Yaskawa INFORM job: DEMO_ROOF_UPPER_0625_3PAINT_68.JBI

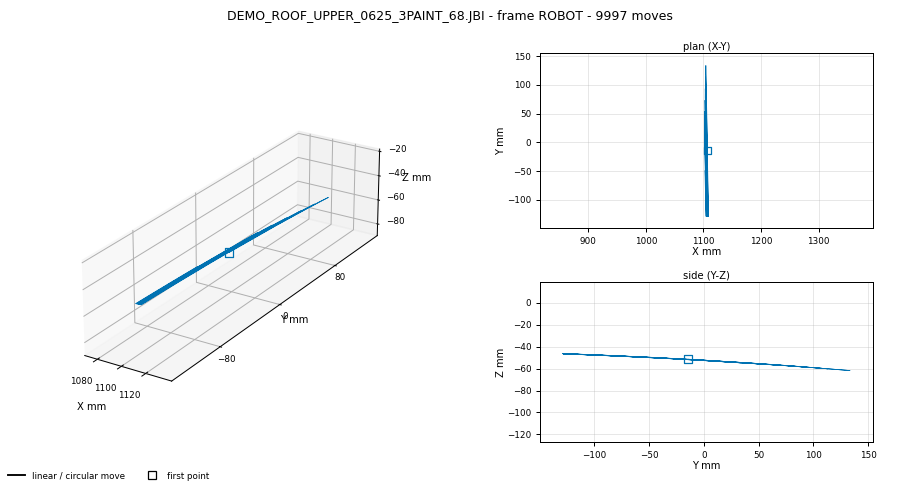
[picture p0: tool path of DEMO_ROOF_UPPER_0625_3PAINT_68.JBI in frame ROBOT, 9997 of 9997 moves have a stored position in this frame; points joined in program order, loops and branches not executed]
/JOB
//NAME DEMO_ROOF_UPPER_0625_3PAINT68
//POS
///NPOS 9997,0,0,0,0,0
///TOOL 0
///USER 0
///POSTYPE ROBOT
///RECTAN
///RCONF 1,0,0,0,0,0,0,0,0,0,0,0,0,0,0,0,0,0,0,0,0,0,0,0
C00000=1106.941,-14.112,-51.375,179.831,6.217,149.173
C00001=1106.936,-13.863,-51.390,179.832,6.222,149.174
C00002=1106.931,-13.614,-51.403,179.832,6.226,149.175
C00003=1106.926,-13.363,-51.417,179.833,6.230,149.176
C00004=1106.921,-13.114,-51.431,179.833,6.235,149.177
C00005=1106.916,-12.865,-51.445,179.834,6.239,149.177
C00006=1106.911,-12.615,-51.459,179.834,6.244,149.178
C00007=1106.906,-12.365,-51.472,179.835,6.249,149.179
C00008=1106.901,-12.115,-51.486,179.836,6.253,149.180
C00009=1106.896,-11.866,-51.500,179.836,6.258,149.181
C00010=1106.891,-11.617,-51.514,179.836,6.262,149.182
C00011=1106.886,-11.367,-51.529,179.837,6.266,149.183
C00012=1106.880,-11.117,-51.542,179.837,6.271,149.183
C00013=1106.876,-10.868,-51.555,179.838,6.276,149.184
C00014=1106.871,-10.618,-51.570,179.839,6.280,149.185
C00015=1106.865,-10.369,-51.584,179.839,6.285,149.186
C00016=1106.860,-10.120,-51.598,179.840,6.290,149.187
C00017=1106.855,-9.870,-51.612,179.840,6.294,149.188
C00018=1106.850,-9.619,-51.626,179.841,6.298,149.188
C00019=1106.845,-9.370,-51.640,179.841,6.303,149.189
C00020=1106.840,-9.121,-51.653,179.842,6.307,149.190
C00021=1106.835,-8.871,-51.668,179.842,6.312,149.191
C00022=1106.830,-8.622,-51.682,179.843,6.316,149.192
C00023=1106.825,-8.373,-51.696,179.844,6.321,149.193
C00024=1106.820,-8.123,-51.710,179.844,6.325,149.194
C00025=1106.815,-7.873,-51.724,179.844,6.330,149.194
C00026=1106.810,-7.623,-51.739,179.845,6.334,149.195
C00027=1106.804,-7.374,-51.753,179.846,6.339,149.196
C00028=1106.800,-7.125,-51.767,179.846,6.344,149.197
C00029=1106.795,-6.875,-51.781,179.847,6.348,149.198
C00030=1106.790,-6.625,-51.794,179.848,6.353,149.198
C00031=1106.785,-6.376,-51.808,179.848,6.357,149.199
C00032=1106.780,-6.126,-51.822,179.848,6.361,149.200
C00033=1106.775,-5.877,-51.837,179.849,6.366,149.201
C00034=1106.770,-5.627,-51.851,179.850,6.370,149.202
C00035=1106.764,-5.378,-51.865,179.850,6.375,149.203
C00036=1106.759,-5.128,-51.879,179.851,6.380,149.204
C00037=1106.756,-4.914,-51.892,179.851,6.383,149.204
C00038=1106.751,-4.700,-51.904,179.852,6.388,149.205
C00039=1106.747,-4.486,-51.916,179.852,6.391,149.206
C00040=1106.742,-4.271,-51.929,179.853,6.395,149.206
C00041=1106.738,-4.057,-51.941,179.853,6.399,149.207
C00042=1106.733,-3.844,-51.953,179.854,6.403,149.208
C00043=1106.729,-3.629,-51.966,179.854,6.406,149.209
C00044=1106.725,-3.415,-51.978,179.855,6.411,149.209
C00045=1106.720,-3.165,-51.992,179.856,6.415,149.210
C00046=1106.715,-2.916,-52.006,179.855,6.419,149.211
C00047=1106.709,-2.667,-52.020,179.856,6.424,149.212
C00048=1106.704,-2.417,-52.034,179.857,6.428,149.213
C00049=1106.699,-2.167,-52.049,179.857,6.433,149.213
C00050=1106.695,-1.918,-52.064,179.858,6.438,149.214
C00051=1106.690,-1.668,-52.078,179.859,6.442,149.215
C00052=1106.685,-1.419,-52.092,179.860,6.447,149.216
C00053=1106.679,-1.169,-52.107,179.860,6.452,149.217
C00054=1106.674,-0.920,-52.121,179.861,6.456,149.217
C00055=1106.669,-0.670,-52.135,179.862,6.461,149.218
C00056=1106.664,-0.421,-52.150,179.862,6.465,149.219
C00057=1106.659,-0.171,-52.165,179.862,6.469,149.220
C00058=1106.654,0.079,-52.179,179.863,6.474,149.221
C00059=1106.649,0.328,-52.193,179.864,6.478,149.222
C00060=1106.644,0.577,-52.208,179.865,6.483,149.222
C00061=1106.640,0.827,-52.222,179.865,6.487,149.223
C00062=1106.633,1.077,-52.237,179.866,6.492,149.224
C00063=1106.628,1.326,-52.251,179.866,6.497,149.225
C00064=1106.624,1.575,-52.266,179.867,6.501,149.226
C00065=1106.619,1.825,-52.280,179.868,6.506,149.227
C00066=1106.614,2.075,-52.295,179.868,6.511,149.227
C00067=1106.609,2.324,-52.310,179.869,6.515,149.228
C00068=1106.603,2.574,-52.325,179.870,6.520,149.229
C00069=1106.598,2.824,-52.339,179.870,6.524,149.230
C00070=1106.594,3.073,-52.354,179.871,6.529,149.231
C00071=1106.589,3.322,-52.368,179.872,6.533,149.231
C00072=1106.584,3.572,-52.382,179.872,6.538,149.232
C00073=1106.578,3.821,-52.398,179.873,6.543,149.233
C00074=1106.574,4.071,-52.412,179.873,6.547,149.234
C00075=1106.569,4.321,-52.427,179.874,6.551,149.235
C00076=1106.564,4.570,-52.442,179.874,6.556,149.236
C00077=1106.559,4.820,-52.456,179.875,6.560,149.237
C00078=1106.554,5.069,-52.471,179.875,6.565,149.237
C00079=1106.549,5.319,-52.486,179.876,6.569,149.238
C00080=1106.544,5.569,-52.500,179.877,6.574,149.239
C00081=1106.539,5.818,-52.515,179.878,6.579,149.240
C00082=1106.533,6.068,-52.530,179.878,6.584,149.241
C00083=1106.529,6.317,-52.545,179.879,6.588,149.241
C00084=1106.524,6.566,-52.559,179.880,6.593,149.242
C00085=1106.518,6.816,-52.575,179.880,6.597,149.243
C00086=1106.513,7.066,-52.589,179.881,6.602,149.244
C00087=1106.509,7.315,-52.604,179.882,6.606,149.245
C00088=1106.503,7.565,-52.619,179.882,6.611,149.246
C00089=1106.498,7.814,-52.634,179.883,6.616,149.247
C00090=1106.493,8.063,-52.648,179.883,6.620,149.247
C00091=1106.488,8.313,-52.664,179.884,6.625,149.248
C00092=1106.483,8.563,-52.678,179.885,6.630,149.249
C00093=1106.479,8.776,-52.691,179.885,6.634,149.250
C00094=1106.474,8.991,-52.704,179.886,6.638,149.251
C00095=1106.470,9.204,-52.716,179.886,6.642,149.251
C00096=1106.466,9.419,-52.729,179.886,6.645,149.252
C00097=1106.461,9.632,-52.742,179.887,6.649,149.253
C00098=1106.458,9.846,-52.755,179.887,6.653,149.254
C00099=1106.453,10.061,-52.768,179.888,6.657,149.254
C00100=1106.449,10.275,-52.781,179.888,6.661,149.255
C00101=1106.444,10.524,-52.795,179.888,6.666,149.256
C00102=1106.439,10.774,-52.811,179.889,6.670,149.257
C00103=1106.434,11.023,-52.826,179.889,6.674,149.258
C00104=1106.428,11.273,-52.841,179.890,6.679,149.259
C00105=1106.424,11.522,-52.856,179.890,6.683,149.259
C00106=1106.418,11.771,-52.871,179.891,6.688,149.260
C00107=1106.413,12.021,-52.886,179.891,6.692,149.261
C00108=1106.409,12.271,-52.901,179.891,6.697,149.262
C00109=1106.404,12.520,-52.917,179.892,6.701,149.263
C00110=1106.399,12.770,-52.931,179.892,6.705,149.264
C00111=1106.394,13.019,-52.946,179.893,6.709,149.265
C00112=1106.389,13.268,-52.961,179.893,6.714,149.265
C00113=1106.383,13.518,-52.976,179.894,6.719,149.266
C00114=1106.379,13.768,-52.991,179.894,6.723,149.267
C00115=1106.373,14.017,-53.007,179.895,6.727,149.268
C00116=1106.369,14.267,-53.022,179.895,6.732,149.269
C00117=1106.364,14.517,-53.037,179.895,6.736,149.270
C00118=1106.359,14.766,-53.052,179.896,6.740,149.270
C00119=1106.354,15.015,-53.068,179.897,6.745,149.271
C00120=1106.349,15.264,-53.083,179.897,6.749,149.272
C00121=1106.343,15.514,-53.098,179.897,6.753,149.273
C00122=1106.339,15.763,-53.113,179.898,6.758,149.274
C00123=1106.334,16.014,-53.129,179.899,6.762,149.274
C00124=1106.329,16.263,-53.143,179.900,6.767,149.275
C00125=1106.324,16.512,-53.159,179.900,6.771,149.276
C00126=1106.319,16.761,-53.174,179.901,6.775,149.277
C00127=1106.314,17.011,-53.190,179.901,6.780,149.278
C00128=1106.309,17.261,-53.204,179.901,6.784,149.279
C00129=1106.304,17.510,-53.220,179.902,6.788,149.279
C00130=1106.299,17.760,-53.235,179.903,6.793,149.280
C00131=1106.294,18.009,-53.250,179.903,6.798,149.281
C00132=1106.289,18.258,-53.266,179.904,6.801,149.282
C00133=1106.284,18.508,-53.281,179.904,6.806,149.283
C00134=1106.279,18.757,-53.297,179.905,6.811,149.284
C00135=1106.274,19.007,-53.313,179.905,6.814,149.284
C00136=1106.269,19.256,-53.328,179.906,6.819,149.285
C00137=1106.264,19.505,-53.343,179.907,6.823,149.286
C00138=1106.260,19.755,-53.359,179.907,6.828,149.287
C00139=1106.254,20.005,-53.374,179.908,6.831,149.287
C00140=1106.249,20.254,-53.390,179.908,6.836,149.288
C00141=1106.244,20.503,-53.405,179.909,6.841,149.289
C00142=1106.239,20.753,-53.421,179.909,6.844,149.290
C00143=1106.234,21.003,-53.436,179.910,6.849,149.291
C00144=1106.229,21.252,-53.451,179.911,6.853,149.291
C00145=1106.224,21.501,-53.467,179.912,6.858,149.292
C00146=1106.219,21.751,-53.483,179.912,6.862,149.293
C00147=1106.215,22.000,-53.498,179.913,6.866,149.294
C00148=1106.209,22.250,-53.513,179.914,6.871,149.294
C00149=1106.205,22.464,-53.527,179.914,6.874,149.295
C00150=1106.201,22.677,-53.540,179.915,6.878,149.296
C00151=1106.196,22.892,-53.554,179.915,6.881,149.296
C00152=1106.192,23.106,-53.567,179.915,6.885,149.297
C00153=1106.188,23.319,-53.580,179.916,6.889,149.298
C00154=1106.184,23.534,-53.594,179.917,6.892,149.298
C00155=1106.179,23.748,-53.607,179.917,6.896,149.299
C00156=1106.175,23.961,-53.620,179.918,6.899,149.300
C00157=1106.170,24.211,-53.636,179.919,6.904,149.300
C00158=1106.165,24.461,-53.652,179.919,6.908,149.301
C00159=1106.160,24.710,-53.667,179.920,6.912,149.302
C00160=1106.156,24.960,-53.683,179.921,6.916,149.302
C00161=1106.150,25.209,-53.698,179.921,6.921,149.303
C00162=1106.145,25.459,-53.714,179.922,6.925,149.304
C00163=1106.140,25.708,-53.730,179.922,6.929,149.305
C00164=1106.136,25.957,-53.745,179.923,6.934,149.306
C00165=1106.130,26.207,-53.761,179.924,6.937,149.306
C00166=1106.126,26.457,-53.777,179.924,6.942,149.307
C00167=1106.120,26.706,-53.793,179.926,6.946,149.308
C00168=1106.115,26.955,-53.809,179.927,6.950,149.308
C00169=1106.111,27.205,-53.824,179.927,6.954,149.309
C00170=1106.106,27.454,-53.840,179.928,6.959,149.310
C00171=1106.100,27.704,-53.855,179.929,6.963,149.311
C00172=1106.096,27.953,-53.872,179.929,6.967,149.311
C00173=1106.090,28.202,-53.888,179.930,6.971,149.312
C00174=1106.085,28.452,-53.903,179.931,6.975,149.313
C00175=1106.081,28.702,-53.919,179.931,6.979,149.313
C00176=1106.076,28.950,-53.935,179.932,6.984,149.314
C00177=1106.071,29.201,-53.951,179.933,6.988,149.315
C00178=1106.066,29.450,-53.966,179.934,6.992,149.316
C00179=1106.061,29.699,-53.983,179.934,6.996,149.316
C00180=1106.056,29.949,-53.999,179.935,7.000,149.317
C00181=1106.050,30.198,-54.014,179.936,7.005,149.318
C00182=1106.046,30.448,-54.031,179.936,7.008,149.318
C00183=1106.041,30.697,-54.046,179.937,7.013,149.319
C00184=1106.037,30.947,-54.062,179.938,7.017,149.320
C00185=1106.031,31.196,-54.078,179.939,7.022,149.321
C00186=1106.026,31.445,-54.094,179.940,7.025,149.321
C00187=1106.021,31.695,-54.110,179.941,7.029,149.322
C00188=1106.016,31.944,-54.126,179.942,7.034,149.323
C00189=1106.011,32.194,-54.142,179.942,7.037,149.323
C00190=1106.006,32.443,-54.158,179.943,7.042,149.324
C00191=1106.002,32.693,-54.174,179.944,7.046,149.325
C00192=1105.996,32.942,-54.191,179.944,7.050,149.326
C00193=1105.991,33.191,-54.206,179.945,7.054,149.326
C00194=1105.987,33.441,-54.223,179.946,7.058,149.327
C00195=1105.981,33.690,-54.238,179.947,7.063,149.327
C00196=1105.976,33.940,-54.254,179.948,7.066,149.328
C00197=1105.971,34.189,-54.271,179.948,7.071,149.329
C00198=1105.967,34.439,-54.287,179.950,7.075,149.330
C00199=1105.961,34.688,-54.303,179.950,7.079,149.330
C00200=1105.957,34.937,-54.320,179.951,7.083,149.331
C00201=1105.952,35.187,-54.335,179.952,7.087,149.332
C00202=1105.947,35.436,-54.352,179.953,7.092,149.332
C00203=1105.942,35.686,-54.367,179.954,7.095,149.333
C00204=1105.937,35.935,-54.384,179.955,7.099,149.334
C00205=1105.933,36.149,-54.398,179.955,7.103,149.334
C00206=1105.928,36.362,-54.412,179.956,7.106,149.335
C00207=1105.924,36.577,-54.426,179.957,7.110,149.335
C00208=1105.920,36.791,-54.439,179.958,7.114,149.336
C00209=1105.916,37.005,-54.454,179.958,7.117,149.336
C00210=1105.911,37.219,-54.467,179.959,7.121,149.337
C00211=1105.907,37.432,-54.482,179.960,7.124,149.338
C00212=1105.903,37.646,-54.495,179.960,7.127,149.338
C00213=1105.898,37.896,-54.512,179.961,7.132,149.339
C00214=1105.893,38.145,-54.528,179.962,7.136,149.340
C00215=1105.888,38.395,-54.544,179.963,7.140,149.340
C00216=1105.883,38.644,-54.560,179.964,7.144,149.341
C00217=1105.879,38.893,-54.577,179.965,7.148,149.341
C00218=1105.873,39.143,-54.594,179.966,7.152,149.342
C00219=1105.868,39.392,-54.610,179.967,7.156,149.343
C00220=1105.864,39.642,-54.627,179.968,7.160,149.343
C00221=1105.858,39.891,-54.642,179.969,7.164,149.344
C00222=1105.854,40.141,-54.659,179.970,7.169,149.345
C00223=1105.849,40.389,-54.675,179.971,7.172,149.345
C00224=1105.844,40.639,-54.691,179.972,7.176,149.346
C00225=1105.839,40.889,-54.708,179.973,7.180,149.347
C00226=1105.834,41.138,-54.725,179.974,7.185,149.347
C00227=1105.829,41.388,-54.741,179.974,7.188,149.348
C00228=1105.824,41.636,-54.758,179.975,7.193,149.348
C00229=1105.819,41.886,-54.774,179.977,7.197,149.349
C00230=1105.814,42.136,-54.791,179.977,7.200,149.350
C00231=1105.809,42.385,-54.807,179.978,7.205,149.350
C00232=1105.804,42.634,-54.824,179.979,7.209,149.351
C00233=1105.799,42.883,-54.840,179.981,7.213,149.352
C00234=1105.794,43.134,-54.857,179.981,7.216,149.352
C00235=1105.789,43.383,-54.873,179.982,7.221,149.353
C00236=1105.784,43.632,-54.890,179.983,7.225,149.353
C00237=1105.780,43.881,-54.906,179.984,7.229,149.354
C00238=1105.775,44.131,-54.924,179.985,7.233,149.355
C00239=1105.770,44.380,-54.940,179.986,7.237,149.355
C00240=1105.765,44.629,-54.957,179.987,7.241,149.356
C00241=1105.761,44.879,-54.973,179.988,7.245,149.357
C00242=1105.754,45.129,-54.989,179.989,7.249,149.357
C00243=1105.750,45.378,-55.006,179.990,7.253,149.358
C00244=1105.745,45.628,-55.023,179.991,7.257,149.359
C00245=1105.740,45.877,-55.040,179.992,7.261,149.359
C00246=1105.735,46.126,-55.056,179.993,7.265,149.360
C00247=1105.731,46.376,-55.073,179.994,7.269,149.360
C00248=1105.726,46.624,-55.089,179.995,7.273,149.361
C00249=1105.720,46.874,-55.107,179.996,7.277,149.362
C00250=1105.716,47.124,-55.123,179.997,7.281,149.362
C00251=1105.711,47.373,-55.140,179.998,7.285,149.363
C00252=1105.706,47.622,-55.157,179.999,7.289,149.363
C00253=1105.701,47.872,-55.174,180.000,7.293,149.364
C00254=1105.696,48.122,-55.191,-179.999,7.297,149.364
C00255=1105.691,48.371,-55.207,-179.997,7.301,149.365
C00256=1105.686,48.620,-55.224,-179.997,7.305,149.366
C00257=1105.681,48.870,-55.241,-179.996,7.309,149.366
C00258=1105.677,49.119,-55.258,-179.994,7.313,149.367
C00259=1105.672,49.367,-55.275,-179.993,7.317,149.367
C00260=1105.667,49.617,-55.292,-179.993,7.321,149.368
C00261=1105.663,49.831,-55.306,-179.991,7.325,149.369
C00262=1105.658,50.045,-55.320,-179.990,7.328,149.369
C00263=1105.654,50.259,-55.335,-179.990,7.331,149.370
C00264=1105.650,50.473,-55.350,-179.989,7.334,149.370
C00265=1105.646,50.687,-55.364,-179.987,7.338,149.371
C00266=1105.642,50.900,-55.378,-179.987,7.342,149.371
C00267=1105.637,51.114,-55.393,-179.986,7.345,149.372
C00268=1105.633,51.328,-55.408,-179.985,7.348,149.372
C00269=1105.628,51.577,-55.424,-179.984,7.352,149.373
C00270=1105.623,51.827,-55.442,-179.982,7.356,149.373
C00271=1105.619,52.075,-55.459,-179.982,7.360,149.374
C00272=1105.613,52.325,-55.476,-179.981,7.364,149.374
C00273=1105.609,52.575,-55.493,-179.979,7.368,149.375
C00274=1105.604,52.825,-55.510,-179.978,7.372,149.376
C00275=1105.599,53.073,-55.527,-179.978,7.376,149.376
C00276=1105.594,53.322,-55.544,-179.976,7.380,149.377
C00277=1105.589,53.572,-55.561,-179.975,7.384,149.377
C00278=1105.584,53.822,-55.578,-179.974,7.388,149.378
C00279=1105.579,54.071,-55.596,-179.972,7.392,149.378
C00280=1105.575,54.320,-55.613,-179.972,7.396,149.379
C00281=1105.569,54.570,-55.630,-179.970,7.400,149.379
C00282=1105.564,54.819,-55.646,-179.969,7.404,149.380
C00283=1105.559,55.068,-55.664,-179.968,7.408,149.381
C00284=1105.555,55.318,-55.681,-179.967,7.411,149.381
C00285=1105.550,55.567,-55.698,-179.966,7.416,149.382
C00286=1105.545,55.816,-55.716,-179.965,7.420,149.382
C00287=1105.540,56.066,-55.733,-179.964,7.424,149.383
C00288=1105.535,56.316,-55.750,-179.963,7.427,149.383
C00289=1105.530,56.564,-55.767,-179.962,7.431,149.384
C00290=1105.525,56.814,-55.785,-179.960,7.436,149.385
C00291=1105.520,57.063,-55.803,-179.959,7.439,149.385
C00292=1105.516,57.313,-55.819,-179.958,7.444,149.386
C00293=1105.510,57.562,-55.836,-179.957,7.447,149.386
C00294=1105.506,57.811,-55.854,-179.956,7.451,149.387
C00295=1105.501,58.061,-55.871,-179.954,7.455,149.387
C00296=1105.496,58.310,-55.889,-179.953,7.459,149.388
C00297=1105.492,58.560,-55.906,-179.952,7.463,149.388
C00298=1105.487,58.809,-55.924,-179.951,7.467,149.389
C00299=1105.481,59.059,-55.941,-179.949,7.471,149.389
C00300=1105.477,59.307,-55.958,-179.948,7.475,149.390
C00301=1105.471,59.557,-55.975,-179.947,7.479,149.391
C00302=1105.467,59.806,-55.993,-179.946,7.482,149.391
C00303=1105.461,60.056,-56.011,-179.945,7.486,149.392
C00304=1105.457,60.304,-56.028,-179.944,7.491,149.392
C00305=1105.452,60.554,-56.045,-179.942,7.495,149.393
C00306=1105.447,60.803,-56.063,-179.941,7.499,149.393
C00307=1105.443,61.053,-56.080,-179.940,7.502,149.394
C00308=1105.438,61.302,-56.098,-179.939,7.506,149.394
C00309=1105.432,61.552,-56.115,-179.937,7.510,149.395
C00310=1105.428,61.801,-56.133,-179.936,7.514,149.396
C00311=1105.423,62.050,-56.150,-179.935,7.518,149.396
C00312=1105.418,62.300,-56.168,-179.934,7.522,149.397
C00313=1105.413,62.549,-56.186,-179.933,7.526,149.397
C00314=1105.408,62.799,-56.203,-179.932,7.530,149.398
C00315=1105.404,63.047,-56.220,-179.930,7.534,149.398
C00316=1105.399,63.297,-56.238,-179.929,7.538,149.399
C00317=1105.394,63.511,-56.253,-179.928,7.541,149.399
C00318=1105.391,63.724,-56.268,-179.927,7.544,149.400
C00319=1105.386,63.938,-56.283,-179.925,7.548,149.400
C00320=1105.382,64.152,-56.298,-179.925,7.551,149.401
C00321=1105.378,64.366,-56.314,-179.924,7.555,149.401
C00322=1105.373,64.580,-56.329,-179.923,7.558,149.401
C00323=1105.370,64.793,-56.344,-179.921,7.562,149.402
C00324=1105.365,65.007,-56.359,-179.920,7.565,149.402
C00325=1105.360,65.256,-56.377,-179.919,7.569,149.403
C00326=1105.356,65.505,-56.395,-179.917,7.573,149.403
C00327=1105.351,65.754,-56.412,-179.917,7.576,149.404
C00328=1105.346,66.004,-56.430,-179.915,7.580,149.404
C00329=1105.341,66.254,-56.448,-179.914,7.584,149.405
C00330=1105.336,66.503,-56.466,-179.913,7.589,149.406
C00331=1105.331,66.752,-56.484,-179.911,7.592,149.406
C00332=1105.326,67.002,-56.501,-179.910,7.597,149.407
C00333=1105.321,67.251,-56.519,-179.909,7.600,149.407
C00334=1105.316,67.500,-56.537,-179.908,7.604,149.408
C00335=1105.312,67.749,-56.555,-179.906,7.608,149.408
C00336=1105.307,67.998,-56.573,-179.905,7.612,149.409
C00337=1105.302,68.247,-56.591,-179.903,7.616,149.409
C00338=1105.297,68.497,-56.608,-179.902,7.620,149.410
C00339=1105.292,68.746,-56.626,-179.901,7.624,149.410
C00340=1105.288,68.996,-56.644,-179.900,7.628,149.411
C00341=1105.283,69.245,-56.662,-179.899,7.631,149.411
C00342=1105.278,69.494,-56.680,-179.897,7.635,149.412
C00343=1105.273,69.744,-56.698,-179.896,7.640,149.412
C00344=1105.268,69.993,-56.716,-179.894,7.644,149.413
C00345=1105.263,70.242,-56.734,-179.893,7.647,149.413
C00346=1105.259,70.491,-56.752,-179.892,7.652,149.414
C00347=1105.254,70.740,-56.770,-179.891,7.655,149.414
C00348=1105.249,70.990,-56.788,-179.889,7.659,149.415
C00349=1105.244,71.239,-56.806,-179.888,7.663,149.415
C00350=1105.239,71.489,-56.824,-179.886,7.667,149.416
C00351=1105.235,71.738,-56.842,-179.885,7.671,149.416
C00352=1105.230,71.987,-56.860,-179.884,7.675,149.417
C00353=1105.225,72.236,-56.878,-179.882,7.679,149.417
C00354=1105.220,72.486,-56.897,-179.881,7.683,149.418
C00355=1105.216,72.735,-56.915,-179.880,7.686,149.418
C00356=1105.210,72.985,-56.933,-179.878,7.690,149.419
C00357=1105.205,73.234,-56.951,-179.877,7.694,149.419
C00358=1105.200,73.483,-56.969,-179.876,7.698,149.420
C00359=1105.196,73.733,-56.988,-179.874,7.702,149.420
C00360=1105.191,73.982,-57.006,-179.873,7.706,149.421
C00361=1105.186,74.231,-57.023,-179.872,7.711,149.421
C00362=1105.181,74.480,-57.041,-179.870,7.714,149.422
C00363=1105.176,74.729,-57.060,-179.868,7.718,149.422
C00364=1105.172,74.979,-57.079,-179.867,7.721,149.423
C00365=1105.166,75.228,-57.097,-179.866,7.726,149.423
C00366=1105.162,75.477,-57.115,-179.865,7.730,149.424
C00367=1105.157,75.727,-57.133,-179.863,7.734,149.424
C00368=1105.152,75.977,-57.151,-179.862,7.738,149.425
C00369=1105.148,76.225,-57.170,-179.860,7.742,149.425
C00370=1105.143,76.474,-57.188,-179.859,7.746,149.426
C00371=1105.137,76.724,-57.207,-179.857,7.750,149.426
C00372=1105.133,76.974,-57.225,-179.856,7.754,149.427
C00373=1105.128,77.187,-57.241,-179.855,7.757,149.427
C00374=1105.124,77.400,-57.256,-179.854,7.760,149.428
C00375=1105.121,77.614,-57.272,-179.853,7.763,149.428
C00376=1105.116,77.828,-57.288,-179.853,7.767,149.429
C00377=1105.112,78.041,-57.303,-179.852,7.770,149.429
C00378=1105.108,78.255,-57.320,-179.851,7.773,149.430
C00379=1105.104,78.468,-57.335,-179.851,7.775,149.430
C00380=1105.100,78.683,-57.351,-179.850,7.778,149.431
C00381=1105.095,78.932,-57.369,-179.848,7.783,149.431
C00382=1105.091,79.180,-57.388,-179.848,7.786,149.432
C00383=1105.085,79.430,-57.407,-179.846,7.790,149.432
C00384=1105.081,79.680,-57.425,-179.846,7.794,149.433
C00385=1105.076,79.928,-57.444,-179.844,7.797,149.433
C00386=1105.071,80.177,-57.462,-179.844,7.801,149.434
C00387=1105.066,80.428,-57.481,-179.842,7.805,149.434
C00388=1105.061,80.676,-57.499,-179.842,7.808,149.435
C00389=1105.056,80.925,-57.517,-179.840,7.812,149.436
C00390=1105.052,81.175,-57.537,-179.839,7.816,149.436
C00391=1105.047,81.424,-57.555,-179.838,7.820,149.437
C00392=1105.042,81.673,-57.573,-179.837,7.824,149.437
C00393=1105.037,81.923,-57.593,-179.836,7.827,149.438
C00394=1105.032,82.172,-57.611,-179.835,7.831,149.438
C00395=1105.028,82.421,-57.629,-179.834,7.834,149.439
C00396=1105.023,82.671,-57.648,-179.833,7.839,149.439
C00397=1105.018,82.919,-57.667,-179.832,7.842,149.440
C00398=1105.014,83.169,-57.685,-179.831,7.846,149.441
C00399=1105.008,83.419,-57.704,-179.830,7.849,149.441
C00400=1105.003,83.667,-57.722,-179.829,7.853,149.442
C00401=1104.999,83.917,-57.741,-179.827,7.857,149.442
C00402=1104.994,84.166,-57.760,-179.826,7.861,149.443
C00403=1104.989,84.415,-57.778,-179.825,7.865,149.443
C00404=1104.984,84.665,-57.798,-179.824,7.868,149.444
C00405=1104.979,84.913,-57.816,-179.823,7.872,149.444
C00406=1104.975,85.163,-57.835,-179.822,7.876,149.445
C00407=1104.970,85.412,-57.854,-179.821,7.879,149.445
C00408=1104.965,85.661,-57.872,-179.819,7.884,149.446
C00409=1104.960,85.911,-57.892,-179.819,7.887,149.446
C00410=1104.955,86.160,-57.910,-179.817,7.891,149.447
C00411=1104.951,86.409,-57.929,-179.816,7.895,149.448
C00412=1104.946,86.658,-57.948,-179.815,7.898,149.448
C00413=1104.942,86.908,-57.966,-179.814,7.902,149.449
C00414=1104.936,87.157,-57.986,-179.813,7.906,149.449
C00415=1104.931,87.406,-58.004,-179.812,7.910,149.450
C00416=1104.927,87.656,-58.023,-179.810,7.914,149.450
C00417=1104.922,87.904,-58.042,-179.809,7.917,149.451
C00418=1104.917,88.154,-58.061,-179.808,7.921,149.451
C00419=1104.912,88.403,-58.080,-179.806,7.925,149.452
C00420=1104.908,88.652,-58.099,-179.805,7.928,149.452
C00421=1104.903,88.902,-58.117,-179.804,7.932,149.453
C00422=1104.898,89.151,-58.137,-179.803,7.936,149.453
C00423=1104.893,89.400,-58.156,-179.802,7.940,149.454
C00424=1104.889,89.649,-58.175,-179.801,7.944,149.454
C00425=1104.884,89.898,-58.193,-179.799,7.947,149.455
C00426=1104.879,90.148,-58.213,-179.798,7.951,149.455
C00427=1104.874,90.397,-58.232,-179.797,7.955,149.456
C00428=1104.870,90.646,-58.251,-179.795,7.959,149.456
C00429=1104.865,90.859,-58.267,-179.794,7.962,149.457
C00430=1104.861,91.074,-58.283,-179.793,7.965,149.457
C00431=1104.857,91.287,-58.300,-179.792,7.968,149.458
C00432=1104.853,91.501,-58.316,-179.791,7.971,149.458
C00433=1104.849,91.714,-58.333,-179.790,7.975,149.458
C00434=1104.845,91.928,-58.349,-179.789,7.978,149.459
C00435=1104.841,92.140,-58.365,-179.788,7.981,149.459
C00436=1104.836,92.355,-58.382,-179.787,7.984,149.460
C00437=1104.831,92.603,-58.401,-179.785,7.988,149.460
C00438=1104.827,92.853,-58.420,-179.784,7.991,149.461
C00439=1104.823,93.102,-58.439,-179.783,7.995,149.461
C00440=1104.817,93.351,-58.459,-179.782,8.000,149.462
C00441=1104.812,93.601,-58.478,-179.780,8.003,149.462
C00442=1104.808,93.850,-58.496,-179.779,8.007,149.463
C00443=1104.803,94.099,-58.516,-179.777,8.010,149.463
C00444=1104.798,94.348,-58.535,-179.776,8.014,149.463
C00445=1104.794,94.597,-58.554,-179.775,8.019,149.464
C00446=1104.788,94.846,-58.574,-179.774,8.022,149.464
C00447=1104.784,95.096,-58.593,-179.772,8.026,149.465
C00448=1104.780,95.345,-58.612,-179.770,8.030,149.465
C00449=1104.774,95.594,-58.632,-179.769,8.033,149.466
C00450=1104.769,95.844,-58.651,-179.768,8.036,149.466
C00451=1104.764,96.092,-58.671,-179.766,8.040,149.467
C00452=1104.760,96.342,-58.690,-179.765,8.045,149.467
C00453=1104.755,96.591,-58.709,-179.764,8.048,149.468
C00454=1104.750,96.840,-58.729,-179.763,8.052,149.468
C00455=1104.746,97.089,-58.748,-179.761,8.056,149.469
C00456=1104.741,97.338,-58.767,-179.759,8.059,149.469
C00457=1104.736,97.588,-58.787,-179.758,8.063,149.469
C00458=1104.731,97.837,-58.806,-179.757,8.066,149.470
C00459=1104.726,98.086,-58.825,-179.755,8.070,149.470
C00460=1104.722,98.336,-58.845,-179.754,8.074,149.471
C00461=1104.717,98.585,-58.864,-179.752,8.078,149.471
C00462=1104.712,98.834,-58.883,-179.751,8.081,149.472
C00463=1104.707,99.083,-58.904,-179.749,8.085,149.472
C00464=1104.703,99.332,-58.923,-179.748,8.089,149.473
C00465=1104.698,99.581,-58.942,-179.746,8.093,149.473
C00466=1104.693,99.831,-58.962,-179.745,8.097,149.473
C00467=1104.688,100.080,-58.982,-179.744,8.100,149.474
C00468=1104.683,100.329,-59.001,-179.742,8.104,149.474
C00469=1104.679,100.578,-59.021,-179.740,8.108,149.475
C00470=1104.675,100.827,-59.040,-179.739,8.111,149.475
C00471=1104.669,101.076,-59.060,-179.737,8.114,149.475
C00472=1104.665,101.326,-59.079,-179.736,8.118,149.476
C00473=1104.660,101.575,-59.099,-179.734,8.122,149.476
C00474=1104.655,101.824,-59.119,-179.733,8.126,149.477
C00475=1104.650,102.073,-59.139,-179.731,8.130,149.477
C00476=1104.645,102.323,-59.158,-179.729,8.134,149.478
C00477=1104.641,102.572,-59.178,-179.728,8.137,149.478
C00478=1104.636,102.820,-59.198,-179.726,8.140,149.478
C00479=1104.632,103.070,-59.217,-179.725,8.144,149.479
C00480=1104.627,103.319,-59.237,-179.723,8.148,149.479
C00481=1104.622,103.568,-59.257,-179.722,8.152,149.480
C00482=1104.617,103.817,-59.276,-179.721,8.155,149.480
C00483=1104.612,104.067,-59.296,-179.718,8.159,149.480
C00484=1104.608,104.316,-59.316,-179.717,8.162,149.481
C00485=1104.604,104.529,-59.334,-179.715,8.165,149.481
C00486=1104.599,104.743,-59.349,-179.714,8.169,149.481
C00487=1104.595,104.957,-59.367,-179.712,8.172,149.482
C00488=1104.591,105.170,-59.384,-179.711,8.175,149.482
C00489=1104.587,105.383,-59.401,-179.710,8.178,149.482
C00490=1104.583,105.597,-59.417,-179.708,8.181,149.483
C00491=1104.579,105.810,-59.435,-179.707,8.184,149.483
C00492=1104.575,106.024,-59.452,-179.706,8.187,149.483
C00493=1104.570,106.272,-59.472,-179.704,8.191,149.484
C00494=1104.566,106.522,-59.491,-179.702,8.195,149.484
C00495=1104.561,106.771,-59.512,-179.700,8.198,149.484
C00496=1104.556,107.020,-59.531,-179.699,8.202,149.485
C00497=1104.552,107.269,-59.552,-179.697,8.205,149.485
C00498=1104.547,107.518,-59.571,-179.696,8.209,149.485
C00499=1104.542,107.767,-59.591,-179.694,8.213,149.486
C00500=1104.537,108.017,-59.612,-179.692,8.216,149.486
C00501=1104.532,108.266,-59.632,-179.690,8.220,149.486
C00502=1104.527,108.515,-59.652,-179.688,8.223,149.487
C00503=1104.523,108.764,-59.672,-179.687,8.227,149.487
C00504=1104.518,109.014,-59.692,-179.685,8.230,149.487
C00505=1104.513,109.262,-59.712,-179.683,8.234,149.487
C00506=1104.508,109.512,-59.731,-179.682,8.237,149.488
C00507=1104.504,109.761,-59.752,-179.680,8.241,149.488
C00508=1104.500,110.010,-59.772,-179.678,8.245,149.489
C00509=1104.494,110.259,-59.792,-179.676,8.248,149.489
C00510=1104.490,110.508,-59.813,-179.674,8.251,149.489
C00511=1104.485,110.757,-59.833,-179.673,8.255,149.489
C00512=1104.480,111.006,-59.852,-179.671,8.258,149.490
C00513=1104.475,111.255,-59.873,-179.669,8.262,149.490
C00514=1104.471,111.504,-59.893,-179.667,8.266,149.490
C00515=1104.466,111.754,-59.913,-179.666,8.268,149.491
C00516=1104.461,112.003,-59.934,-179.664,8.272,149.491
C00517=1104.457,112.252,-59.954,-179.662,8.276,149.491
C00518=1104.452,112.501,-59.974,-179.661,8.279,149.492
C00519=1104.448,112.750,-59.994,-179.659,8.282,149.492
C00520=1104.442,113.000,-60.015,-179.657,8.286,149.492
C00521=1104.438,113.249,-60.036,-179.656,8.289,149.493
C00522=1104.433,113.498,-60.055,-179.654,8.293,149.493
C00523=1104.429,113.747,-60.076,-179.652,8.296,149.493
C00524=1104.423,113.996,-60.096,-179.651,8.299,149.494
C00525=1104.419,114.245,-60.117,-179.649,8.303,149.494
C00526=1104.414,114.494,-60.136,-179.647,8.307,149.494
C00527=1104.409,114.743,-60.157,-179.646,8.309,149.494
C00528=1104.404,114.992,-60.178,-179.644,8.313,149.495
C00529=1104.400,115.241,-60.198,-179.642,8.317,149.495
C00530=1104.395,115.490,-60.218,-179.641,8.319,149.495
C00531=1104.390,115.740,-60.239,-179.639,8.323,149.496
C00532=1104.385,115.989,-60.259,-179.637,8.327,149.496
C00533=1104.381,116.238,-60.279,-179.635,8.329,149.496
C00534=1104.376,116.487,-60.300,-179.633,8.333,149.496
C00535=1104.371,116.736,-60.321,-179.632,8.337,149.497
C00536=1104.367,116.985,-60.341,-179.630,8.340,149.497
C00537=1104.362,117.235,-60.362,-179.628,8.343,149.497
C00538=1104.357,117.483,-60.382,-179.627,8.347,149.498
C00539=1104.353,117.732,-60.403,-179.625,8.350,149.498
C00540=1104.348,117.982,-60.424,-179.623,8.353,149.498
C00541=1104.344,118.195,-60.440,-179.622,8.356,149.498
C00542=1104.340,118.408,-60.459,-179.621,8.359,149.499
C00543=1104.336,118.622,-60.476,-179.619,8.362,149.499
C00544=1104.332,118.835,-60.494,-179.617,8.365,149.499
C00545=1104.328,119.049,-60.512,-179.616,8.368,149.500
C00546=1104.324,119.262,-60.530,-179.614,8.371,149.500
C00547=1104.320,119.476,-60.546,-179.613,8.373,149.500
C00548=1104.316,119.688,-60.564,-179.612,8.376,149.500
C00549=1104.311,119.938,-60.586,-179.609,8.380,149.500
C00550=1104.307,120.187,-60.606,-179.608,8.383,149.501
C00551=1104.302,120.436,-60.627,-179.606,8.386,149.501
C00552=1104.297,120.685,-60.647,-179.604,8.390,149.501
C00553=1104.292,120.935,-60.668,-179.603,8.393,149.502
C00554=1104.288,121.183,-60.689,-179.601,8.396,149.502
C00555=1104.283,121.432,-60.709,-179.599,8.400,149.502
C00556=1104.278,121.681,-60.731,-179.598,8.402,149.502
C00557=1104.274,121.930,-60.751,-179.596,8.406,149.503
C00558=1104.269,122.179,-60.772,-179.594,8.410,149.503
C00559=1104.264,122.428,-60.792,-179.593,8.413,149.503
C00560=1104.260,122.678,-60.814,-179.591,8.416,149.504
C00561=1104.255,122.927,-60.834,-179.589,8.420,149.504
C00562=1104.250,123.176,-60.856,-179.588,8.423,149.504
C00563=1104.246,123.425,-60.876,-179.585,8.426,149.505
C00564=1104.241,123.674,-60.897,-179.583,8.430,149.505
C00565=1104.236,123.923,-60.917,-179.582,8.434,149.505
C00566=1104.231,124.172,-60.938,-179.580,8.436,149.505
C00567=1104.227,124.422,-60.960,-179.578,8.440,149.506
C00568=1104.222,124.670,-60.981,-179.577,8.444,149.506
C00569=1104.217,124.920,-61.002,-179.575,8.446,149.506
C00570=1104.213,125.169,-61.022,-179.573,8.450,149.507
C00571=1104.208,125.417,-61.044,-179.571,8.453,149.507
C00572=1104.203,125.666,-61.064,-179.570,8.456,149.507
C00573=1104.199,125.916,-61.086,-179.568,8.460,149.507
C00574=1104.194,126.165,-61.107,-179.566,8.463,149.508
C00575=1104.190,126.414,-61.128,-179.565,8.466,149.508
C00576=1104.184,126.663,-61.149,-179.562,8.470,149.508
C00577=1104.180,126.911,-61.170,-179.561,8.474,149.509
C00578=1104.176,127.161,-61.191,-179.559,8.476,149.509
C00579=1104.170,127.411,-61.212,-179.557,8.480,149.509
C00580=1104.166,127.659,-61.233,-179.555,8.483,149.509
C00581=1104.161,127.908,-61.254,-179.554,8.486,149.510
C00582=1104.156,128.157,-61.275,-179.552,8.490,149.510
C00583=1104.152,128.406,-61.296,-179.550,8.493,149.510
C00584=1104.147,128.656,-61.317,-179.549,8.496,149.510
C00585=1104.142,128.904,-61.339,-179.547,8.500,149.511
C00586=1104.137,129.154,-61.360,-179.545,8.503,149.511
C00587=1104.133,129.402,-61.381,-179.544,8.506,149.511
C00588=1104.129,129.652,-61.403,-179.541,8.510,149.512
C00589=1104.124,129.901,-61.424,-179.540,8.513,149.512
C00590=1104.119,130.150,-61.445,-179.538,8.517,149.512
C00591=1104.114,130.398,-61.466,-179.536,8.520,149.512
C00592=1104.110,130.648,-61.488,-179.534,8.523,149.513
C00593=1104.105,130.897,-61.509,-179.533,8.527,149.513
C00594=1104.101,131.146,-61.530,-179.531,8.530,149.513
C00595=1104.096,131.395,-61.552,-179.529,8.533,149.514
C00596=1104.091,131.644,-61.573,-179.527,8.537,149.514
C00597=1104.087,131.878,-61.592,-179.526,8.539,149.514
C00598=1104.083,132.113,-61.613,-179.524,8.543,149.514
C00599=1104.078,132.348,-61.633,-179.523,8.546,149.515
C00600=1104.073,132.582,-61.653,-179.520,8.550,149.515
C00601=1104.069,132.816,-61.673,-179.519,8.552,149.515
C00602=1104.065,133.051,-61.694,-179.517,8.556,149.515
C00603=1104.060,133.285,-61.714,-179.516,8.559,149.516
C00604=1104.056,133.520,-61.734,-179.514,8.562,149.516
C00605=1103.825,123.405,-60.927,-179.583,8.428,149.504
C00606=1103.830,123.156,-60.906,-179.585,8.424,149.504
C00607=1103.835,122.908,-60.885,-179.586,8.421,149.503
C00608=1103.839,122.658,-60.864,-179.588,8.418,149.503
C00609=1103.844,122.409,-60.843,-179.590,8.414,149.503
C00610=1103.849,122.160,-60.822,-179.591,8.411,149.503
C00611=1103.853,121.911,-60.802,-179.593,8.408,149.502
C00612=1103.858,121.662,-60.781,-179.595,8.404,149.502
C00613=1103.863,121.413,-60.760,-179.596,8.401,149.502
C00614=1103.868,121.164,-60.739,-179.599,8.398,149.502
C00615=1103.872,120.915,-60.718,-179.600,8.394,149.501
C00616=1103.877,120.666,-60.697,-179.602,8.391,149.501
C00617=1103.881,120.416,-60.677,-179.604,8.388,149.501
C00618=1103.886,120.167,-60.656,-179.605,8.384,149.500
C00619=1103.891,119.918,-60.635,-179.607,8.381,149.500
C00620=1103.895,119.669,-60.615,-179.609,8.378,149.500
C00621=1103.900,119.420,-60.594,-179.611,8.374,149.500
C00622=1103.907,119.061,-60.564,-179.613,8.370,149.499
C00623=1103.914,118.704,-60.535,-179.615,8.365,149.499
C00624=1103.921,118.345,-60.505,-179.618,8.360,149.498
C00625=1103.928,117.987,-60.476,-179.620,8.355,149.498
C00626=1103.932,117.738,-60.455,-179.622,8.352,149.498
C00627=1103.937,117.488,-60.434,-179.624,8.349,149.497
C00628=1103.942,117.239,-60.414,-179.626,8.345,149.497
C00629=1103.946,116.990,-60.394,-179.627,8.342,149.497
C00630=1103.951,116.741,-60.373,-179.629,8.338,149.496
C00631=1103.956,116.492,-60.352,-179.631,8.335,149.496
C00632=1103.960,116.243,-60.332,-179.632,8.332,149.496
C00633=1103.965,115.994,-60.311,-179.634,8.328,149.496
C00634=1103.970,115.745,-60.291,-179.636,8.324,149.495
C00635=1103.974,115.496,-60.270,-179.637,8.322,149.495
C00636=1103.980,115.246,-60.250,-179.639,8.318,149.494
C00637=1103.984,114.997,-60.230,-179.641,8.314,149.494
C00638=1103.989,114.748,-60.209,-179.642,8.312,149.494
C00639=1103.993,114.499,-60.189,-179.644,8.308,149.494
C00640=1103.998,114.250,-60.168,-179.646,8.304,149.493
C00641=1104.003,114.001,-60.148,-179.647,8.302,149.493
C00642=1104.007,113.752,-60.128,-179.649,8.298,149.493
C00643=1104.013,113.502,-60.107,-179.651,8.294,149.492
C00644=1104.017,113.253,-60.087,-179.652,8.291,149.492
C00645=1104.021,113.005,-60.066,-179.654,8.288,149.492
C00646=1104.026,112.755,-60.047,-179.656,8.284,149.492
C00647=1104.031,112.506,-60.026,-179.657,8.281,149.491
C00648=1104.036,112.257,-60.005,-179.659,8.277,149.491
C00649=1104.041,112.008,-59.985,-179.661,8.274,149.490
C00650=1104.046,111.759,-59.966,-179.662,8.271,149.490
C00651=1104.050,111.510,-59.945,-179.664,8.267,149.490
C00652=1104.055,111.261,-59.924,-179.666,8.263,149.490
C00653=1104.060,111.011,-59.905,-179.667,8.261,149.489
C00654=1104.064,110.762,-59.884,-179.669,8.257,149.489
C00655=1104.069,110.513,-59.864,-179.671,8.253,149.489
C00656=1104.074,110.264,-59.844,-179.673,8.250,149.488
C00657=1104.078,110.015,-59.824,-179.675,8.246,149.488
C00658=1104.084,109.766,-59.804,-179.677,8.242,149.488
C00659=1104.089,109.517,-59.784,-179.678,8.240,149.488
C00660=1104.093,109.268,-59.763,-179.680,8.236,149.487
C00661=1104.098,109.018,-59.743,-179.682,8.232,149.487
C00662=1104.102,108.769,-59.723,-179.683,8.228,149.486
C00663=1104.107,108.520,-59.703,-179.686,8.225,149.486
C00664=1104.111,108.271,-59.683,-179.687,8.221,149.486
C00665=1104.117,108.022,-59.664,-179.689,8.218,149.486
C00666=1104.121,107.773,-59.643,-179.690,8.215,149.485
C00667=1104.126,107.524,-59.623,-179.692,8.211,149.485
C00668=1104.130,107.274,-59.603,-179.694,8.207,149.484
C00669=1104.135,107.025,-59.583,-179.695,8.203,149.484
C00670=1104.140,106.775,-59.563,-179.697,8.200,149.484
C00671=1104.146,106.527,-59.543,-179.698,8.197,149.483
C00672=1104.150,106.278,-59.523,-179.701,8.193,149.483
C00673=1104.155,106.028,-59.503,-179.702,8.189,149.483
C00674=1104.158,105.815,-59.487,-179.704,8.187,149.482
C00675=1104.163,105.602,-59.470,-179.705,8.183,149.482
C00676=1104.167,105.388,-59.453,-179.707,8.180,149.482
C00677=1104.171,105.174,-59.435,-179.708,8.177,149.481
C00678=1104.174,104.961,-59.419,-179.709,8.174,149.481
C00679=1104.179,104.748,-59.402,-179.711,8.170,149.481
C00680=1104.183,104.534,-59.385,-179.712,8.167,149.480
C00681=1104.187,104.320,-59.367,-179.713,8.165,149.480
C00682=1104.192,104.072,-59.347,-179.715,8.161,149.480
C00683=1104.197,103.823,-59.328,-179.717,8.157,149.479
C00684=1104.202,103.573,-59.308,-179.718,8.153,149.479
C00685=1104.205,103.324,-59.288,-179.719,8.150,149.478
C00686=1104.211,103.076,-59.269,-179.721,8.147,149.478
C00687=1104.215,102.826,-59.249,-179.723,8.143,149.478
C00688=1104.220,102.577,-59.229,-179.725,8.139,149.477
C00689=1104.224,102.327,-59.209,-179.726,8.135,149.477
C00690=1104.230,102.079,-59.190,-179.727,8.132,149.477
C00691=1104.235,101.829,-59.170,-179.729,8.128,149.476
C00692=1104.239,101.580,-59.150,-179.731,8.124,149.476
C00693=1104.244,101.331,-59.130,-179.732,8.120,149.475
C00694=1104.249,101.082,-59.111,-179.734,8.117,149.475
C00695=1104.254,100.832,-59.091,-179.735,8.113,149.475
C00696=1104.258,100.583,-59.072,-179.737,8.110,149.474
C00697=1104.263,100.335,-59.052,-179.738,8.106,149.474
C00698=1104.268,100.085,-59.033,-179.740,8.102,149.473
C00699=1104.272,99.835,-59.013,-179.741,8.098,149.473
C00700=1104.278,99.587,-58.994,-179.742,8.095,149.472
C00701=1104.282,99.338,-58.973,-179.744,8.091,149.472
C00702=1104.286,99.088,-58.954,-179.746,8.087,149.471
C00703=1104.291,98.840,-58.935,-179.747,8.083,149.471
C00704=1104.296,98.590,-58.915,-179.748,8.080,149.471
C00705=1104.301,98.340,-58.896,-179.750,8.076,149.470
C00706=1104.306,98.092,-58.876,-179.751,8.072,149.470
C00707=1104.310,97.842,-58.857,-179.753,8.068,149.469
C00708=1104.315,97.593,-58.838,-179.754,8.065,149.469
C00709=1104.320,97.344,-58.818,-179.756,8.061,149.468
C00710=1104.325,97.094,-58.799,-179.757,8.058,149.468
C00711=1104.329,96.845,-58.780,-179.759,8.054,149.468
C00712=1104.334,96.597,-58.760,-179.760,8.051,149.467
C00713=1104.339,96.347,-58.740,-179.761,8.047,149.467
C00714=1104.344,96.098,-58.721,-179.763,8.043,149.466
C00715=1104.348,95.849,-58.702,-179.764,8.039,149.466
C00716=1104.353,95.599,-58.682,-179.765,8.036,149.465
C00717=1104.358,95.351,-58.663,-179.767,8.031,149.465
C00718=1104.363,95.101,-58.644,-179.768,8.028,149.464
C00719=1104.368,94.852,-58.625,-179.770,8.024,149.464
C00720=1104.373,94.602,-58.605,-179.771,8.021,149.463
C00721=1104.378,94.353,-58.586,-179.772,8.017,149.463
C00722=1104.382,94.104,-58.567,-179.774,8.013,149.463
C00723=1104.387,93.855,-58.547,-179.775,8.009,149.462
C00724=1104.392,93.606,-58.528,-179.776,8.005,149.461
C00725=1104.396,93.356,-58.509,-179.778,8.002,149.461
C00726=1104.402,93.108,-58.490,-179.779,7.998,149.461
C00727=1104.406,92.858,-58.471,-179.780,7.994,149.460
C00728=1104.411,92.610,-58.451,-179.781,7.990,149.459
C00729=1104.416,92.360,-58.432,-179.783,7.986,149.459
C00730=1104.419,92.146,-58.416,-179.784,7.983,149.459
C00731=1104.424,91.933,-58.399,-179.785,7.980,149.458
C00732=1104.427,91.719,-58.383,-179.786,7.977,149.458
C00733=1104.433,91.505,-58.367,-179.787,7.974,149.457
C00734=1104.436,91.292,-58.350,-179.788,7.970,149.457
C00735=1104.440,91.078,-58.334,-179.789,7.967,149.456
C00736=1104.444,90.865,-58.317,-179.790,7.964,149.456
C00737=1104.448,90.652,-58.302,-179.791,7.961,149.456
C00738=1104.453,90.402,-58.282,-179.793,7.957,149.455
C00739=1104.458,90.153,-58.263,-179.794,7.954,149.455
C00740=1104.463,89.904,-58.244,-179.795,7.949,149.454
C00741=1104.467,89.655,-58.226,-179.797,7.946,149.454
C00742=1104.472,89.405,-58.206,-179.798,7.942,149.453
C00743=1104.478,89.156,-58.187,-179.799,7.938,149.453
C00744=1104.482,88.907,-58.168,-179.800,7.934,149.452
C00745=1104.487,88.658,-58.149,-179.801,7.931,149.452
C00746=1104.491,88.408,-58.130,-179.802,7.927,149.451
C00747=1104.497,88.159,-58.111,-179.804,7.923,149.451
C00748=1104.501,87.910,-58.092,-179.805,7.920,149.450
C00749=1104.506,87.661,-58.073,-179.806,7.916,149.449
C00750=1104.511,87.412,-58.054,-179.808,7.912,149.449
C00751=1104.516,87.162,-58.035,-179.808,7.908,149.448
C00752=1104.520,86.913,-58.017,-179.810,7.904,149.448
C00753=1104.524,86.664,-57.998,-179.811,7.901,149.448
C00754=1104.530,86.415,-57.979,-179.812,7.897,149.447
C00755=1104.534,86.165,-57.960,-179.814,7.893,149.446
C00756=1104.540,85.916,-57.941,-179.814,7.890,149.446
C00757=1104.544,85.667,-57.923,-179.816,7.886,149.445
C00758=1104.549,85.418,-57.903,-179.817,7.881,149.445
C00759=1104.554,85.169,-57.885,-179.818,7.878,149.444
C00760=1104.559,84.919,-57.865,-179.819,7.874,149.444
C00761=1104.564,84.670,-57.847,-179.820,7.871,149.443
C00762=1104.568,84.421,-57.828,-179.821,7.867,149.443
C00763=1104.573,84.171,-57.810,-179.822,7.864,149.442
C00764=1104.578,83.923,-57.791,-179.824,7.860,149.442
C00765=1104.583,83.672,-57.772,-179.825,7.855,149.441
C00766=1104.588,83.424,-57.753,-179.826,7.852,149.441
C00767=1104.592,83.175,-57.736,-179.827,7.848,149.440
C00768=1104.597,82.925,-57.716,-179.828,7.845,149.440
C00769=1104.602,82.676,-57.698,-179.829,7.841,149.439
C00770=1104.606,82.427,-57.679,-179.830,7.838,149.438
C00771=1104.612,82.177,-57.660,-179.831,7.833,149.438
C00772=1104.616,81.929,-57.642,-179.833,7.829,149.437
C00773=1104.621,81.679,-57.623,-179.833,7.826,149.437
C00774=1104.626,81.430,-57.604,-179.834,7.822,149.436
C00775=1104.631,81.181,-57.586,-179.835,7.818,149.436
C00776=1104.635,80.931,-57.568,-179.836,7.814,149.435
C00777=1104.641,80.682,-57.548,-179.837,7.811,149.435
C00778=1104.646,80.433,-57.530,-179.838,7.807,149.434
C00779=1104.650,80.183,-57.511,-179.839,7.804,149.433
C00780=1104.655,79.934,-57.493,-179.840,7.799,149.433
C00781=1104.660,79.685,-57.475,-179.841,7.796,149.432
C00782=1104.664,79.436,-57.456,-179.843,7.792,149.432
C00783=1104.669,79.186,-57.438,-179.843,7.789,149.431
C00784=1104.675,78.937,-57.419,-179.845,7.785,149.431
C00785=1104.679,78.688,-57.400,-179.845,7.781,149.430
C00786=1104.683,78.474,-57.384,-179.846,7.778,149.430
C00787=1104.688,78.261,-57.369,-179.847,7.775,149.429
C00788=1104.691,78.047,-57.352,-179.848,7.772,149.429
C00789=1104.696,77.833,-57.337,-179.849,7.769,149.428
C00790=1104.699,77.620,-57.322,-179.849,7.765,149.428
C00791=1104.703,77.406,-57.305,-179.850,7.762,149.427
C00792=1104.708,77.193,-57.290,-179.851,7.759,149.427
C00793=1104.712,76.979,-57.274,-179.852,7.756,149.426
C00794=1104.716,76.730,-57.256,-179.854,7.752,149.426
C00795=1104.721,76.480,-57.238,-179.855,7.748,149.425
C00796=1104.727,76.231,-57.219,-179.857,7.744,149.425
C00797=1104.732,75.982,-57.201,-179.858,7.740,149.424
C00798=1104.736,75.732,-57.182,-179.859,7.736,149.424
C00799=1104.741,75.483,-57.164,-179.860,7.732,149.423
C00800=1104.746,75.234,-57.146,-179.862,7.729,149.423
C00801=1104.751,74.985,-57.128,-179.863,7.725,149.422
C00802=1104.756,74.735,-57.109,-179.865,7.720,149.422
C00803=1104.760,74.486,-57.090,-179.866,7.716,149.421
C00804=1104.765,74.237,-57.073,-179.868,7.713,149.421
C00805=1104.770,73.988,-57.055,-179.869,7.708,149.420
C00806=1104.774,73.738,-57.036,-179.870,7.704,149.420
C00807=1104.779,73.489,-57.018,-179.872,7.700,149.419
C00808=1104.784,73.240,-57.000,-179.872,7.697,149.419
C00809=1104.789,72.990,-56.982,-179.874,7.693,149.418
C00810=1104.795,72.741,-56.964,-179.876,7.689,149.418
C00811=1104.799,72.491,-56.945,-179.877,7.685,149.417
C00812=1104.804,72.242,-56.927,-179.878,7.681,149.417
C00813=1104.809,71.993,-56.909,-179.880,7.677,149.416
C00814=1104.814,71.744,-56.891,-179.881,7.673,149.416
C00815=1104.818,71.495,-56.873,-179.883,7.669,149.415
C00816=1104.823,71.246,-56.855,-179.884,7.666,149.415
C00817=1104.828,70.996,-56.836,-179.885,7.662,149.414
C00818=1104.833,70.747,-56.818,-179.886,7.658,149.414
C00819=1104.838,70.497,-56.801,-179.888,7.654,149.413
C00820=1104.843,70.248,-56.783,-179.889,7.649,149.413
C00821=1104.848,69.999,-56.765,-179.890,7.646,149.412
C00822=1104.853,69.749,-56.747,-179.892,7.642,149.412
C00823=1104.857,69.500,-56.729,-179.893,7.638,149.411
C00824=1104.862,69.250,-56.711,-179.894,7.634,149.411
C00825=1104.867,69.001,-56.693,-179.896,7.630,149.410
C00826=1104.872,68.752,-56.675,-179.897,7.626,149.409
C00827=1104.876,68.503,-56.657,-179.898,7.622,149.409
C00828=1104.881,68.254,-56.639,-179.900,7.618,149.409
C00829=1104.886,68.004,-56.621,-179.901,7.614,149.408
C00830=1104.891,67.755,-56.603,-179.902,7.611,149.408
C00831=1104.896,67.506,-56.586,-179.903,7.607,149.407
C00832=1104.901,67.256,-56.568,-179.905,7.603,149.406
C00833=1104.906,67.006,-56.549,-179.906,7.599,149.406
C00834=1104.910,66.758,-56.532,-179.907,7.594,149.405
C00835=1104.915,66.508,-56.514,-179.909,7.591,149.405
C00836=1104.920,66.259,-56.496,-179.909,7.587,149.404
C00837=1104.925,66.009,-56.479,-179.911,7.583,149.404
C00838=1104.930,65.760,-56.461,-179.913,7.579,149.403
C00839=1104.935,65.511,-56.443,-179.914,7.575,149.403
C00840=1104.940,65.262,-56.425,-179.915,7.571,149.402
C00841=1104.945,65.012,-56.408,-179.916,7.567,149.402
C00842=1104.949,64.799,-56.392,-179.917,7.564,149.401
C00843=1104.953,64.585,-56.377,-179.918,7.561,149.401
C00844=1104.956,64.371,-56.362,-179.919,7.557,149.400
C00845=1104.961,64.157,-56.347,-179.921,7.553,149.400
C00846=1104.965,63.944,-56.332,-179.922,7.550,149.399
C00847=1104.969,63.730,-56.317,-179.923,7.547,149.399
C00848=1104.973,63.517,-56.302,-179.924,7.543,149.399
C00849=1104.978,63.303,-56.287,-179.925,7.540,149.398
C00850=1104.983,63.054,-56.269,-179.926,7.536,149.398
C00851=1104.988,62.804,-56.251,-179.927,7.533,149.397
C00852=1104.992,62.555,-56.234,-179.928,7.529,149.396
C00853=1104.997,62.306,-56.216,-179.930,7.525,149.396
C00854=1105.002,62.056,-56.199,-179.931,7.520,149.395
C00855=1105.007,61.807,-56.181,-179.932,7.516,149.395
C00856=1105.012,61.558,-56.163,-179.933,7.513,149.394
C00857=1105.017,61.308,-56.146,-179.934,7.509,149.394
C00858=1105.022,61.059,-56.128,-179.936,7.505,149.393
C00859=1105.027,60.809,-56.111,-179.937,7.501,149.393
C00860=1105.031,60.561,-56.093,-179.939,7.497,149.392
C00861=1105.036,60.311,-56.076,-179.939,7.493,149.392
C00862=1105.041,60.062,-56.058,-179.941,7.490,149.391
C00863=1105.046,59.812,-56.040,-179.942,7.485,149.391
C00864=1105.050,59.563,-56.024,-179.943,7.481,149.390
C00865=1105.055,59.314,-56.006,-179.945,7.477,149.389
C00866=1105.061,59.064,-55.988,-179.945,7.474,149.389
C00867=1105.065,58.815,-55.971,-179.947,7.470,149.388
C00868=1105.070,58.565,-55.954,-179.948,7.465,149.388
C00869=1105.075,58.316,-55.936,-179.949,7.461,149.387
C00870=1105.079,58.067,-55.919,-179.950,7.457,149.387
C00871=1105.085,57.817,-55.902,-179.951,7.454,149.386
C00872=1105.089,57.568,-55.884,-179.952,7.450,149.386
C00873=1105.095,57.319,-55.867,-179.954,7.446,149.385
C00874=1105.099,57.070,-55.849,-179.955,7.441,149.384
C00875=1105.105,56.820,-55.832,-179.956,7.438,149.384
C00876=1105.109,56.571,-55.815,-179.957,7.434,149.383
C00877=1105.114,56.321,-55.798,-179.958,7.430,149.383
C00878=1105.119,56.071,-55.780,-179.960,7.426,149.382
C00879=1105.123,55.823,-55.763,-179.961,7.422,149.382
C00880=1105.129,55.573,-55.746,-179.962,7.418,149.381
C00881=1105.134,55.324,-55.729,-179.963,7.414,149.381
C00882=1105.139,55.075,-55.711,-179.964,7.410,149.380
C00883=1105.144,54.825,-55.694,-179.965,7.406,149.379
C00884=1105.148,54.576,-55.677,-179.966,7.402,149.379
C00885=1105.153,54.326,-55.659,-179.967,7.399,149.378
C00886=1105.158,54.077,-55.643,-179.969,7.394,149.378
C00887=1105.163,53.827,-55.626,-179.970,7.390,149.377
C00888=1105.168,53.578,-55.609,-179.971,7.387,149.377
C00889=1105.173,53.329,-55.591,-179.972,7.383,149.376
C00890=1105.177,53.080,-55.575,-179.973,7.379,149.376
C00891=1105.183,52.830,-55.557,-179.974,7.374,149.375
C00892=1105.187,52.580,-55.541,-179.975,7.371,149.374
C00893=1105.193,52.332,-55.523,-179.976,7.367,149.374
C00894=1105.197,52.082,-55.506,-179.977,7.363,149.373
C00895=1105.202,51.833,-55.489,-179.979,7.358,149.372
C00896=1105.207,51.583,-55.472,-179.979,7.355,149.372
C00897=1105.212,51.334,-55.454,-179.981,7.351,149.371
C00898=1105.216,51.120,-55.440,-179.981,7.348,149.371
C00899=1105.220,50.906,-55.426,-179.983,7.343,149.370
C00900=1105.225,50.692,-55.411,-179.984,7.340,149.370
C00901=1105.229,50.478,-55.397,-179.984,7.337,149.369
C00902=1105.233,50.265,-55.382,-179.985,7.334,149.369
C00903=1105.237,50.051,-55.368,-179.986,7.331,149.368
C00904=1105.242,49.838,-55.353,-179.987,7.327,149.368
C00905=1105.246,49.624,-55.339,-179.988,7.324,149.367
C00906=1105.251,49.374,-55.322,-179.989,7.319,149.367
C00907=1105.256,49.125,-55.305,-179.990,7.316,149.366
C00908=1105.260,48.876,-55.288,-179.991,7.311,149.365
C00909=1105.266,48.627,-55.271,-179.993,7.308,149.365
C00910=1105.270,48.377,-55.254,-179.994,7.303,149.364
C00911=1105.275,48.128,-55.237,-179.994,7.300,149.364
C00912=1105.280,47.878,-55.220,-179.995,7.295,149.363
C00913=1105.285,47.629,-55.204,-179.997,7.292,149.363
C00914=1105.289,47.380,-55.187,-179.998,7.287,149.362
C00915=1105.295,47.130,-55.170,-179.998,7.284,149.361
C00916=1105.299,46.880,-55.153,-179.999,7.279,149.361
C00917=1105.304,46.632,-55.137,179.999,7.275,149.360
C00918=1105.309,46.382,-55.120,179.999,7.272,149.360
C00919=1105.314,46.132,-55.103,179.998,7.268,149.359
C00920=1105.319,45.883,-55.087,179.997,7.263,149.358
C00921=1105.324,45.634,-55.069,179.995,7.259,149.358
C00922=1105.329,45.384,-55.053,179.995,7.256,149.357
C00923=1105.334,45.135,-55.036,179.993,7.252,149.357
C00924=1105.339,44.886,-55.019,179.992,7.247,149.356
C00925=1105.343,44.636,-55.003,179.991,7.243,149.355
C00926=1105.348,44.386,-54.987,179.991,7.240,149.355
C00927=1105.354,44.137,-54.970,179.989,7.236,149.354
C00928=1105.359,43.887,-54.953,179.988,7.231,149.353
C00929=1105.363,43.638,-54.936,179.988,7.228,149.353
C00930=1105.368,43.389,-54.920,179.987,7.224,149.352
C00931=1105.373,43.139,-54.903,179.986,7.219,149.352
C00932=1105.378,42.891,-54.886,179.985,7.215,149.351
C00933=1105.383,42.641,-54.870,179.984,7.211,149.350
C00934=1105.388,42.391,-54.854,179.983,7.207,149.350
C00935=1105.394,42.142,-54.837,179.981,7.203,149.349
C00936=1105.398,41.892,-54.820,179.981,7.200,149.348
C00937=1105.402,41.643,-54.804,179.980,7.195,149.348
C00938=1105.408,41.394,-54.787,179.979,7.191,149.347
C00939=1105.412,41.144,-54.771,179.978,7.187,149.347
C00940=1105.418,40.895,-54.754,179.977,7.183,149.346
C00941=1105.423,40.645,-54.738,179.976,7.179,149.345
C00942=1105.427,40.396,-54.721,179.975,7.175,149.345
C00943=1105.432,40.147,-54.705,179.975,7.171,149.344
C00944=1105.437,39.897,-54.689,179.974,7.167,149.343
C00945=1105.443,39.648,-54.672,179.973,7.163,149.343
C00946=1105.447,39.399,-54.655,179.971,7.158,149.342
C00947=1105.452,39.148,-54.639,179.971,7.155,149.341
C00948=1105.457,38.900,-54.623,179.969,7.151,149.341
C00949=1105.462,38.650,-54.606,179.968,7.146,149.340
C00950=1105.467,38.401,-54.591,179.968,7.143,149.340
C00951=1105.472,38.151,-54.574,179.967,7.139,149.339
C00952=1105.477,37.902,-54.558,179.966,7.134,149.338
C00953=1105.482,37.652,-54.541,179.965,7.130,149.338
C00954=1105.486,37.438,-54.527,179.964,7.127,149.337
C00955=1105.491,37.225,-54.513,179.964,7.123,149.336
C00956=1105.495,37.011,-54.499,179.963,7.120,149.336
C00957=1105.499,36.797,-54.486,179.962,7.116,149.335
C00958=1105.503,36.583,-54.472,179.962,7.113,149.335
C00959=1105.507,36.369,-54.458,179.960,7.109,149.334
C00960=1105.511,36.156,-54.444,179.960,7.105,149.333
C00961=1105.516,35.942,-54.430,179.959,7.102,149.333
C00962=1105.520,35.692,-54.413,179.958,7.098,149.332
C00963=1105.526,35.443,-54.398,179.958,7.094,149.332
C00964=1105.530,35.193,-54.381,179.957,7.090,149.331
C00965=1105.536,34.944,-54.365,179.956,7.085,149.330
C00966=1105.541,34.694,-54.348,179.955,7.081,149.329
C00967=1105.546,34.445,-54.332,179.954,7.078,149.329
C00968=1105.551,34.195,-54.316,179.953,7.073,149.328
C00969=1105.556,33.946,-54.300,179.952,7.069,149.327
C00970=1105.560,33.696,-54.284,179.952,7.066,149.327
C00971=1105.565,33.448,-54.267,179.951,7.061,149.326
C00972=1105.570,33.197,-54.252,179.950,7.057,149.325
C00973=1105.575,32.949,-54.235,179.949,7.053,149.325
C00974=1105.580,32.699,-54.219,179.949,7.049,149.324
C00975=1105.586,32.449,-54.204,179.948,7.044,149.323
C00976=1105.591,32.200,-54.187,179.947,7.040,149.323
C00977=1105.595,31.951,-54.172,179.946,7.037,149.322
C00978=1105.600,31.702,-54.156,179.945,7.032,149.321
C00979=1105.605,31.452,-54.140,179.944,7.028,149.321
C00980=1105.610,31.203,-54.123,179.944,7.024,149.320
C00981=1105.614,30.953,-54.107,179.943,7.020,149.319
C00982=1105.620,30.703,-54.092,179.942,7.015,149.318
C00983=1105.624,30.454,-54.075,179.941,7.012,149.318
C00984=1105.630,30.205,-54.060,179.941,7.007,149.317
C00985=1105.635,29.955,-54.044,179.940,7.003,149.316
C00986=1105.639,29.706,-54.027,179.939,6.999,149.316
C00987=1105.645,29.456,-54.012,179.938,6.995,149.315
C00988=1105.650,29.206,-53.996,179.937,6.991,149.314
C00989=1105.654,28.958,-53.980,179.937,6.986,149.313
C00990=1105.659,28.708,-53.965,179.936,6.983,149.313
C00991=1105.664,28.458,-53.949,179.935,6.978,149.312
C00992=1105.669,28.209,-53.932,179.935,6.974,149.311
C00993=1105.674,27.959,-53.916,179.934,6.970,149.311
C00994=1105.679,27.710,-53.901,179.933,6.966,149.310
C00995=1105.685,27.461,-53.884,179.932,6.961,149.309
C00996=1105.689,27.211,-53.869,179.931,6.957,149.308
C00997=1105.694,26.962,-53.853,179.931,6.953,149.308
C00998=1105.699,26.713,-53.838,179.930,6.949,149.307
C00999=1105.704,26.463,-53.821,179.929,6.944,149.306
C01000=1105.709,26.214,-53.806,179.929,6.941,149.306
C01001=1105.715,25.964,-53.790,179.928,6.936,149.305
C01002=1105.719,25.714,-53.775,179.927,6.932,149.304
C01003=1105.724,25.465,-53.759,179.927,6.928,149.303
C01004=1105.729,25.216,-53.743,179.926,6.923,149.302
C01005=1105.734,24.966,-53.727,179.925,6.919,149.302
C01006=1105.739,24.717,-53.712,179.925,6.916,149.301
C01007=1105.744,24.468,-53.696,179.924,6.911,149.300
C01008=1105.749,24.218,-53.680,179.923,6.907,149.300
C01009=1105.754,23.968,-53.665,179.923,6.902,149.299
C01010=1105.758,23.754,-53.652,179.922,6.898,149.298
C01011=1105.763,23.541,-53.638,179.922,6.895,149.297
C01012=1105.767,23.326,-53.625,179.921,6.891,149.297
C01013=1105.770,23.112,-53.611,179.921,6.888,149.296
C01014=1105.775,22.899,-53.598,179.920,6.885,149.296
C01015=1105.780,22.684,-53.584,179.919,6.880,149.295
C01016=1105.783,22.470,-53.571,179.919,6.877,149.294
C01017=1105.788,22.257,-53.558,179.918,6.873,149.294
C01018=1105.793,22.006,-53.542,179.918,6.869,149.293
C01019=1105.797,21.758,-53.526,179.917,6.865,149.292
C01020=1105.803,21.509,-53.511,179.917,6.860,149.291
C01021=1105.808,21.259,-53.495,179.915,6.856,149.291
C01022=1105.813,21.009,-53.479,179.916,6.852,149.290
C01023=1105.817,20.760,-53.464,179.915,6.847,149.289
C01024=1105.823,20.511,-53.449,179.914,6.843,149.288
C01025=1105.827,20.262,-53.434,179.913,6.838,149.287
C01026=1105.832,20.011,-53.418,179.913,6.835,149.287
C01027=1105.838,19.762,-53.402,179.912,6.830,149.286
C01028=1105.842,19.513,-53.387,179.911,6.826,149.285
C01029=1105.848,19.264,-53.371,179.911,6.822,149.284
C01030=1105.852,19.013,-53.356,179.911,6.817,149.283
C01031=1105.857,18.764,-53.341,179.910,6.813,149.283
C01032=1105.863,18.514,-53.326,179.909,6.808,149.282
C01033=1105.868,18.265,-53.310,179.909,6.805,149.281
C01034=1105.873,18.016,-53.295,179.908,6.800,149.280
C01035=1105.878,17.766,-53.279,179.908,6.795,149.279
C01036=1105.882,17.517,-53.264,179.907,6.792,149.279
C01037=1105.888,17.267,-53.249,179.907,6.787,149.278
C01038=1105.892,17.018,-53.234,179.906,6.782,149.277
C01039=1105.898,16.769,-53.218,179.906,6.779,149.276
C01040=1105.902,16.519,-53.202,179.905,6.774,149.275
C01041=1105.907,16.269,-53.188,179.905,6.770,149.274
C01042=1105.913,16.020,-53.172,179.903,6.765,149.274
C01043=1105.917,15.770,-53.157,179.904,6.761,149.273
C01044=1105.923,15.521,-53.142,179.903,6.757,149.272
C01045=1105.927,15.271,-53.126,179.902,6.752,149.271
C01046=1105.932,15.022,-53.111,179.902,6.748,149.270
C01047=1105.937,14.772,-53.096,179.901,6.744,149.270
C01048=1105.943,14.523,-53.081,179.901,6.739,149.269
C01049=1105.947,14.274,-53.066,179.900,6.734,149.268
C01050=1105.953,14.024,-53.050,179.900,6.731,149.267
C01051=1105.957,13.775,-53.035,179.899,6.726,149.266
C01052=1105.962,13.524,-53.020,179.899,6.721,149.265
C01053=1105.967,13.275,-53.005,179.899,6.717,149.264
C01054=1105.972,13.026,-52.989,179.898,6.713,149.264
C01055=1105.977,12.777,-52.974,179.897,6.708,149.263
C01056=1105.983,12.527,-52.959,179.897,6.704,149.262
C01057=1105.987,12.278,-52.944,179.897,6.700,149.261
C01058=1105.993,12.028,-52.929,179.896,6.695,149.260
C01059=1105.998,11.779,-52.915,179.896,6.690,149.259
C01060=1106.003,11.528,-52.899,179.896,6.686,149.259
C01061=1106.007,11.279,-52.884,179.895,6.682,149.258
C01062=1106.012,11.030,-52.869,179.895,6.677,149.257
C01063=1106.018,10.780,-52.854,179.894,6.673,149.256
C01064=1106.022,10.531,-52.839,179.894,6.669,149.255
C01065=1106.028,10.281,-52.824,179.893,6.664,149.254
C01066=1106.031,10.067,-52.811,179.893,6.660,149.253
C01067=1106.036,9.854,-52.798,179.893,6.657,149.253
C01068=1106.040,9.639,-52.785,179.892,6.652,149.252
C01069=1106.044,9.426,-52.772,179.892,6.648,149.251
C01070=1106.049,9.211,-52.759,179.891,6.645,149.251
C01071=1106.053,8.997,-52.747,179.891,6.641,149.250
C01072=1106.058,8.783,-52.735,179.891,6.637,149.249
C01073=1106.062,8.569,-52.721,179.890,6.633,149.248
C01074=1106.067,8.319,-52.707,179.889,6.628,149.247
C01075=1106.072,8.070,-52.691,179.889,6.624,149.247
C01076=1106.077,7.821,-52.676,179.888,6.619,149.246
C01077=1106.082,7.571,-52.662,179.888,6.614,149.245
C01078=1106.087,7.322,-52.646,179.887,6.610,149.244
C01079=1106.092,7.072,-52.632,179.886,6.605,149.243
C01080=1106.097,6.823,-52.617,179.886,6.601,149.242
C01081=1106.102,6.573,-52.603,179.885,6.596,149.241
C01082=1106.107,6.324,-52.587,179.885,6.591,149.241
C01083=1106.112,6.074,-52.573,179.884,6.587,149.240
C01084=1106.117,5.825,-52.558,179.883,6.582,149.239
C01085=1106.122,5.575,-52.543,179.883,6.577,149.238
C01086=1106.127,5.326,-52.528,179.882,6.573,149.237
C01087=1106.132,5.076,-52.514,179.881,6.568,149.237
C01088=1106.137,4.827,-52.499,179.880,6.564,149.236
C01089=1106.142,4.577,-52.484,179.880,6.559,149.235
C01090=1106.147,4.327,-52.469,179.879,6.554,149.234
C01091=1106.152,4.078,-52.454,179.878,6.550,149.233
C01092=1106.157,3.829,-52.440,179.878,6.545,149.232
C01093=1106.162,3.579,-52.425,179.877,6.541,149.231
C01094=1106.167,3.330,-52.410,179.876,6.536,149.231
C01095=1106.172,3.080,-52.396,179.876,6.531,149.230
C01096=1106.177,2.831,-52.381,179.875,6.527,149.229
C01097=1106.182,2.581,-52.367,179.875,6.523,149.228
C01098=1106.188,2.331,-52.352,179.874,6.519,149.227
C01099=1106.192,2.082,-52.337,179.874,6.514,149.227
C01100=1106.197,1.832,-52.323,179.873,6.509,149.226
C01101=1106.202,1.582,-52.308,179.873,6.504,149.225
C01102=1106.207,1.333,-52.293,179.872,6.500,149.224
C01103=1106.212,1.083,-52.279,179.871,6.495,149.223
C01104=1106.217,0.834,-52.264,179.871,6.491,149.222
C01105=1106.223,0.585,-52.250,179.870,6.486,149.222
C01106=1106.228,0.336,-52.235,179.869,6.482,149.221
C01107=1106.233,0.086,-52.221,179.869,6.477,149.220
C01108=1106.237,-0.164,-52.207,179.868,6.472,149.219
C01109=1106.242,-0.414,-52.192,179.867,6.468,149.218
C01110=1106.247,-0.663,-52.177,179.867,6.463,149.217
C01111=1106.253,-0.913,-52.163,179.866,6.458,149.217
C01112=1106.258,-1.162,-52.148,179.866,6.455,149.216
C01113=1106.263,-1.412,-52.134,179.865,6.450,149.215
C01114=1106.268,-1.661,-52.120,179.865,6.445,149.214
C01115=1106.273,-1.910,-52.105,179.864,6.441,149.213
C01116=1106.278,-2.160,-52.091,179.863,6.436,149.213
C01117=1106.283,-2.410,-52.077,179.862,6.432,149.212
C01118=1106.288,-2.659,-52.062,179.862,6.427,149.211
C01119=1106.293,-2.909,-52.048,179.861,6.423,149.210
C01120=1106.298,-3.159,-52.034,179.860,6.418,149.209
C01121=1106.303,-3.407,-52.019,179.860,6.413,149.208
C01122=1106.307,-3.622,-52.007,179.860,6.410,149.208
C01123=1106.312,-3.836,-51.994,179.859,6.406,149.207
C01124=1106.316,-4.050,-51.982,179.858,6.402,149.206
C01125=1106.320,-4.265,-51.970,179.858,6.398,149.206
C01126=1106.325,-4.479,-51.958,179.858,6.394,149.205
C01127=1106.329,-4.692,-51.946,179.857,6.390,149.204
C01128=1106.333,-4.907,-51.933,179.856,6.386,149.203
C01129=1106.338,-5.121,-51.921,179.856,6.383,149.203
C01130=1106.343,-5.371,-51.907,179.856,6.378,149.202
C01131=1106.347,-5.620,-51.893,179.855,6.374,149.201
C01132=1106.353,-5.869,-51.879,179.854,6.369,149.200
C01133=1106.358,-6.119,-51.864,179.854,6.364,149.199
C01134=1106.363,-6.369,-51.850,179.853,6.360,149.198
C01135=1106.368,-6.619,-51.836,179.853,6.355,149.198
C01136=1106.373,-6.868,-51.822,179.852,6.352,149.197
C01137=1106.378,-7.117,-51.808,179.852,6.347,149.196
C01138=1106.383,-7.367,-51.793,179.851,6.342,149.195
C01139=1106.388,-7.617,-51.779,179.851,6.337,149.194
C01140=1106.393,-7.866,-51.765,179.850,6.333,149.194
C01141=1106.399,-8.115,-51.751,179.849,6.328,149.193
C01142=1106.404,-8.365,-51.737,179.849,6.324,149.192
C01143=1106.408,-8.615,-51.723,179.848,6.319,149.191
C01144=1106.413,-8.864,-51.709,179.848,6.315,149.190
C01145=1106.418,-9.113,-51.695,179.847,6.311,149.189
C01146=1106.423,-9.363,-51.681,179.847,6.306,149.188
C01147=1106.428,-9.613,-51.666,179.846,6.301,149.187
C01148=1106.434,-9.863,-51.653,179.845,6.297,149.187
C01149=1106.439,-10.112,-51.639,179.845,6.292,149.186
C01150=1106.444,-10.362,-51.625,179.844,6.287,149.185
C01151=1106.448,-10.611,-51.611,179.844,6.283,149.184
C01152=1106.453,-10.861,-51.597,179.843,6.279,149.183
C01153=1106.459,-11.110,-51.583,179.843,6.274,149.183
C01154=1106.464,-11.360,-51.568,179.842,6.270,149.182
C01155=1106.469,-11.610,-51.555,179.842,6.265,149.181
C01156=1106.475,-11.859,-51.541,179.841,6.260,149.180
C01157=1106.479,-12.108,-51.527,179.840,6.256,149.179
C01158=1106.484,-12.358,-51.513,179.840,6.252,149.178
C01159=1106.490,-12.608,-51.500,179.840,6.247,149.177
C01160=1106.495,-12.857,-51.485,179.839,6.243,149.177
C01161=1106.500,-13.107,-51.471,179.839,6.238,149.176
C01162=1106.504,-13.356,-51.458,179.838,6.233,149.175
C01163=1106.509,-13.605,-51.444,179.837,6.229,149.174
C01164=1106.515,-13.856,-51.430,179.838,6.225,149.173
C01165=1106.520,-14.105,-51.416,179.837,6.220,149.172
C01166=1106.524,-14.354,-51.402,179.837,6.215,149.171
C01167=1106.530,-14.605,-51.389,179.836,6.211,149.170
C01168=1106.535,-14.854,-51.375,179.836,6.206,149.170
C01169=1106.540,-15.103,-51.361,179.835,6.202,149.169
C01170=1106.545,-15.353,-51.348,179.834,6.197,149.168
C01171=1106.550,-15.602,-51.334,179.834,6.193,149.167
C01172=1106.555,-15.852,-51.320,179.834,6.188,149.166
C01173=1106.560,-16.102,-51.307,179.833,6.184,149.165
C01174=1106.565,-16.351,-51.293,179.833,6.179,149.164
C01175=1106.570,-16.601,-51.278,179.832,6.174,149.163
C01176=1106.576,-16.850,-51.265,179.832,6.169,149.163
C01177=1106.580,-17.100,-51.252,179.831,6.165,149.162
C01178=1106.585,-17.314,-51.239,179.831,6.161,149.161
C01179=1106.590,-17.528,-51.228,179.830,6.158,149.160
C01180=1106.594,-17.742,-51.216,179.831,6.154,149.159
C01181=1106.598,-17.957,-51.204,179.830,6.149,149.159
C01182=1106.602,-18.171,-51.193,179.830,6.145,149.158
C01183=1106.606,-18.385,-51.181,179.829,6.142,149.157
C01184=1106.611,-18.600,-51.170,179.828,6.137,149.157
C01185=1106.616,-18.813,-51.158,179.829,6.134,149.156
C01186=1106.620,-19.063,-51.145,179.828,6.129,149.155
C01187=1106.626,-19.312,-51.131,179.828,6.124,149.154
C01188=1106.631,-19.563,-51.117,179.827,6.119,149.153
C01189=1106.636,-19.812,-51.104,179.827,6.115,149.152
C01190=1106.641,-20.062,-51.090,179.827,6.111,149.151
C01191=1106.646,-20.312,-51.076,179.826,6.106,149.150
C01192=1106.651,-20.561,-51.063,179.826,6.101,149.149
C01193=1106.656,-20.811,-51.049,179.825,6.097,149.148
C01194=1106.661,-21.060,-51.037,179.825,6.092,149.147
C01195=1106.666,-21.310,-51.022,179.824,6.087,149.147
C01196=1106.671,-21.559,-51.010,179.824,6.083,149.146
C01197=1106.676,-21.809,-50.995,179.824,6.078,149.145
C01198=1106.682,-22.058,-50.982,179.823,6.074,149.144
C01199=1106.686,-22.308,-50.969,179.823,6.069,149.143
C01200=1106.692,-22.557,-50.955,179.822,6.064,149.142
C01201=1106.697,-22.807,-50.942,179.822,6.060,149.141
C01202=1106.702,-23.056,-50.928,179.822,6.055,149.140
C01203=1106.707,-23.306,-50.915,179.822,6.050,149.139
C01204=1106.712,-23.555,-50.902,179.822,6.046,149.138
C01205=1106.717,-23.805,-50.889,179.821,6.041,149.137
C01206=1106.723,-24.055,-50.875,179.821,6.036,149.136
C01207=1106.727,-24.304,-50.862,179.820,6.032,149.136
C01208=1106.733,-24.554,-50.849,179.820,6.027,149.135
C01209=1106.737,-24.804,-50.836,179.820,6.022,149.133
C01210=1106.743,-25.053,-50.822,179.819,6.017,149.133
C01211=1106.747,-25.303,-50.809,179.819,6.013,149.132
C01212=1106.753,-25.553,-50.796,179.819,6.008,149.131
C01213=1106.758,-25.801,-50.782,179.818,6.004,149.130
C01214=1106.763,-26.052,-50.769,179.818,5.999,149.129
C01215=1106.768,-26.301,-50.756,179.819,5.995,149.128
C01216=1106.774,-26.551,-50.742,179.818,5.990,149.127
C01217=1106.779,-26.800,-50.729,179.818,5.985,149.126
C01218=1106.784,-27.050,-50.716,179.818,5.981,149.125
C01219=1106.789,-27.300,-50.703,179.818,5.976,149.124
C01220=1106.793,-27.550,-50.690,179.818,5.972,149.123
C01221=1106.799,-27.799,-50.676,179.818,5.967,149.122
C01222=1106.804,-28.048,-50.664,179.818,5.962,149.121
C01223=1106.809,-28.298,-50.650,179.818,5.958,149.120
C01224=1106.815,-28.548,-50.637,179.817,5.954,149.119
C01225=1106.819,-28.797,-50.624,179.817,5.949,149.118
C01226=1106.825,-29.047,-50.610,179.817,5.945,149.117
C01227=1106.829,-29.297,-50.597,179.816,5.940,149.117
C01228=1106.835,-29.546,-50.584,179.817,5.936,149.116
C01229=1106.840,-29.796,-50.572,179.816,5.932,149.115
C01230=1106.845,-30.046,-50.559,179.816,5.927,149.114
C01231=1106.850,-30.295,-50.545,179.816,5.923,149.113
C01232=1106.855,-30.544,-50.532,179.815,5.918,149.112
C01233=1106.860,-30.794,-50.519,179.815,5.913,149.111
C01234=1106.865,-31.009,-50.508,179.815,5.910,149.110
C01235=1106.869,-31.223,-50.497,179.815,5.906,149.109
C01236=1106.873,-31.437,-50.486,179.814,5.902,149.109
C01237=1106.878,-31.651,-50.474,179.814,5.898,149.108
C01238=1106.882,-31.866,-50.463,179.814,5.895,149.107
C01239=1106.887,-32.080,-50.452,179.814,5.891,149.106
C01240=1106.891,-32.294,-50.441,179.814,5.887,149.106
C01241=1106.895,-32.509,-50.430,179.813,5.883,149.105
C01242=1106.901,-32.758,-50.417,179.813,5.879,149.104
C01243=1106.905,-33.008,-50.404,179.813,5.874,149.103
C01244=1106.911,-33.258,-50.391,179.812,5.870,149.102
C01245=1106.916,-33.507,-50.378,179.812,5.866,149.101
C01246=1106.920,-33.757,-50.365,179.812,5.861,149.100
C01247=1106.925,-34.006,-50.352,179.811,5.856,149.099
C01248=1106.931,-34.256,-50.339,179.811,5.853,149.099
C01249=1106.936,-34.506,-50.326,179.811,5.848,149.098
C01250=1106.941,-34.755,-50.313,179.810,5.843,149.097
C01251=1106.946,-35.004,-50.301,179.810,5.839,149.096
C01252=1106.952,-35.254,-50.288,179.810,5.835,149.095
C01253=1106.956,-35.504,-50.275,179.809,5.830,149.094
C01254=1106.962,-35.753,-50.262,179.809,5.825,149.093
C01255=1106.967,-36.003,-50.250,179.809,5.820,149.092
C01256=1106.972,-36.253,-50.237,179.808,5.816,149.092
C01257=1106.977,-36.503,-50.224,179.808,5.812,149.091
C01258=1106.983,-36.752,-50.211,179.807,5.807,149.090
C01259=1106.988,-37.001,-50.199,179.807,5.803,149.089
C01260=1106.992,-37.251,-50.186,179.806,5.798,149.088
C01261=1106.998,-37.501,-50.173,179.806,5.793,149.087
C01262=1107.003,-37.750,-50.160,179.805,5.788,149.086
C01263=1107.008,-38.000,-50.147,179.806,5.785,149.085
C01264=1107.013,-38.250,-50.134,179.805,5.780,149.084
C01265=1107.018,-38.499,-50.122,179.805,5.775,149.084
C01266=1107.024,-38.749,-50.109,179.804,5.770,149.083
C01267=1107.029,-38.999,-50.096,179.804,5.766,149.082
C01268=1107.034,-39.249,-50.084,179.803,5.761,149.081
C01269=1107.039,-39.498,-50.071,179.803,5.756,149.080
C01270=1107.044,-39.747,-50.059,179.803,5.751,149.079
C01271=1107.049,-39.997,-50.046,179.802,5.747,149.078
C01272=1107.054,-40.247,-50.034,179.802,5.742,149.077
C01273=1107.059,-40.496,-50.021,179.802,5.737,149.076
C01274=1107.065,-40.746,-50.008,179.801,5.732,149.075
C01275=1107.070,-40.995,-49.995,179.801,5.727,149.074
C01276=1107.075,-41.245,-49.983,179.800,5.723,149.073
C01277=1107.080,-41.495,-49.971,179.800,5.718,149.072
C01278=1107.085,-41.745,-49.958,179.800,5.713,149.071
C01279=1107.090,-41.994,-49.945,179.800,5.708,149.070
C01280=1107.095,-42.243,-49.933,179.799,5.702,149.069
C01281=1107.101,-42.493,-49.921,179.798,5.698,149.068
C01282=1107.105,-42.743,-49.908,179.798,5.693,149.067
C01283=1107.110,-42.993,-49.895,179.798,5.688,149.066
C01284=1107.116,-43.243,-49.883,179.798,5.683,149.065
C01285=1107.121,-43.492,-49.871,179.798,5.678,149.064
C01286=1107.126,-43.741,-49.858,179.799,5.674,149.063
C01287=1107.132,-43.991,-49.846,179.799,5.669,149.062
C01288=1107.136,-44.241,-49.833,179.799,5.664,149.061
C01289=1107.141,-44.490,-49.821,179.799,5.660,149.060
C01290=1107.146,-44.706,-49.810,179.800,5.656,149.059
C01291=1107.151,-44.919,-49.800,179.800,5.652,149.058
C01292=1107.155,-45.133,-49.789,179.799,5.647,149.057
C01293=1107.160,-45.348,-49.778,179.799,5.643,149.056
C01294=1107.164,-45.563,-49.768,179.800,5.639,149.055
C01295=1107.168,-45.777,-49.757,179.800,5.635,149.054
C01296=1107.172,-45.991,-49.746,179.800,5.631,149.053
C01297=1107.178,-46.206,-49.736,179.800,5.628,149.052
C01298=1107.182,-46.456,-49.723,179.800,5.622,149.051
C01299=1107.187,-46.705,-49.710,179.801,5.618,149.050
C01300=1107.192,-46.955,-49.699,179.800,5.613,149.049
C01301=1107.197,-47.204,-49.687,179.801,5.608,149.048
C01302=1107.203,-47.454,-49.675,179.801,5.604,149.047
C01303=1107.208,-47.703,-49.662,179.801,5.599,149.046
C01304=1107.213,-47.953,-49.649,179.801,5.594,149.045
C01305=1107.218,-48.203,-49.638,179.801,5.590,149.044
C01306=1107.223,-48.452,-49.625,179.802,5.585,149.043
C01307=1107.228,-48.703,-49.613,179.802,5.581,149.042
C01308=1107.233,-48.952,-49.600,179.802,5.576,149.040
C01309=1107.239,-49.202,-49.588,179.802,5.570,149.039
C01310=1107.244,-49.451,-49.576,179.802,5.566,149.038
C01311=1107.249,-49.701,-49.564,179.802,5.561,149.037
C01312=1107.255,-49.950,-49.551,179.802,5.556,149.036
C01313=1107.259,-50.200,-49.540,179.803,5.552,149.035
C01314=1107.264,-50.449,-49.527,179.802,5.547,149.034
C01315=1107.270,-50.699,-49.515,179.803,5.542,149.033
C01316=1107.275,-50.949,-49.503,179.803,5.538,149.032
C01317=1107.280,-51.198,-49.491,179.803,5.533,149.031
C01318=1107.286,-51.448,-49.479,179.803,5.529,149.030
C01319=1107.291,-51.698,-49.466,179.804,5.523,149.029
C01320=1107.296,-51.948,-49.455,179.803,5.519,149.028
C01321=1107.301,-52.197,-49.443,179.804,5.514,149.026
C01322=1107.306,-52.447,-49.431,179.804,5.509,149.025
C01323=1107.311,-52.696,-49.418,179.804,5.505,149.024
C01324=1107.317,-52.946,-49.406,179.804,5.500,149.023
C01325=1107.321,-53.197,-49.394,179.804,5.495,149.022
C01326=1107.327,-53.446,-49.381,179.804,5.490,149.021
C01327=1107.331,-53.695,-49.370,179.805,5.486,149.020
C01328=1107.337,-53.945,-49.358,179.805,5.481,149.019
C01329=1107.342,-54.195,-49.346,179.804,5.476,149.018
C01330=1107.347,-54.445,-49.334,179.805,5.472,149.017
C01331=1107.352,-54.694,-49.322,179.805,5.467,149.016
C01332=1107.357,-54.944,-49.310,179.805,5.462,149.015
C01333=1107.363,-55.194,-49.298,179.805,5.458,149.014
C01334=1107.368,-55.443,-49.285,179.805,5.453,149.013
C01335=1107.373,-55.693,-49.273,179.806,5.449,149.011
C01336=1107.378,-55.942,-49.262,179.806,5.443,149.010
C01337=1107.383,-56.192,-49.250,179.805,5.439,149.009
C01338=1107.388,-56.442,-49.238,179.806,5.434,149.008
C01339=1107.394,-56.692,-49.226,179.806,5.430,149.007
C01340=1107.398,-56.941,-49.214,179.806,5.424,149.006
C01341=1107.404,-57.190,-49.202,179.806,5.420,149.005
C01342=1107.410,-57.440,-49.190,179.806,5.415,149.004
C01343=1107.414,-57.689,-49.179,179.806,5.410,149.003
C01344=1107.420,-57.939,-49.167,179.807,5.406,149.002
C01345=1107.425,-58.189,-49.155,179.806,5.401,149.001
C01346=1107.429,-58.404,-49.145,179.807,5.397,149.000
C01347=1107.434,-58.618,-49.135,179.807,5.393,148.999
C01348=1107.438,-58.833,-49.124,179.807,5.389,148.998
C01349=1107.443,-59.047,-49.114,179.807,5.385,148.997
C01350=1107.447,-59.262,-49.104,179.807,5.381,148.996
C01351=1107.451,-59.476,-49.093,179.807,5.377,148.995
C01352=1107.456,-59.690,-49.084,179.807,5.373,148.994
C01353=1107.460,-59.905,-49.074,179.807,5.369,148.993
C01354=1107.466,-60.155,-49.062,179.807,5.364,148.992
C01355=1107.470,-60.404,-49.050,179.807,5.359,148.992
C01356=1107.475,-60.654,-49.038,179.806,5.355,148.991
C01357=1107.481,-60.904,-49.026,179.806,5.349,148.989
C01358=1107.486,-61.153,-49.015,179.805,5.344,148.989
C01359=1107.491,-61.403,-49.003,179.805,5.339,148.988
C01360=1107.497,-61.652,-48.991,179.805,5.334,148.986
C01361=1107.502,-61.902,-48.980,179.805,5.329,148.986
C01362=1107.507,-62.152,-48.968,179.805,5.324,148.984
C01363=1107.511,-62.401,-48.956,179.804,5.319,148.983
C01364=1107.517,-62.651,-48.944,179.804,5.315,148.982
C01365=1107.522,-62.901,-48.933,179.804,5.310,148.981
C01366=1107.527,-63.151,-48.921,179.804,5.305,148.980
C01367=1107.532,-63.401,-48.909,179.803,5.299,148.979
C01368=1107.538,-63.649,-48.898,179.803,5.294,148.978
C01369=1107.543,-63.899,-48.887,179.803,5.289,148.977
C01370=1107.548,-64.149,-48.875,179.803,5.284,148.976
C01371=1107.553,-64.399,-48.863,179.803,5.279,148.975
C01372=1107.558,-64.649,-48.852,179.802,5.274,148.974
C01373=1107.563,-64.898,-48.840,179.802,5.269,148.973
C01374=1107.569,-65.148,-48.828,179.802,5.264,148.972
C01375=1107.574,-65.397,-48.817,179.802,5.259,148.971
C01376=1107.580,-65.647,-48.805,179.802,5.254,148.970
C01377=1107.584,-65.897,-48.794,179.801,5.249,148.969
C01378=1107.590,-66.147,-48.782,179.801,5.243,148.968
C01379=1107.594,-66.396,-48.771,179.801,5.239,148.967
C01380=1107.600,-66.646,-48.759,179.801,5.234,148.966
C01381=1107.605,-66.895,-48.748,179.801,5.228,148.964
C01382=1107.611,-67.145,-48.736,179.801,5.224,148.963
C01383=1107.615,-67.395,-48.725,179.801,5.219,148.962
C01384=1107.621,-67.645,-48.714,179.801,5.213,148.961
C01385=1107.626,-67.894,-48.703,179.801,5.209,148.960
C01386=1107.631,-68.144,-48.692,179.801,5.203,148.959
C01387=1107.636,-68.394,-48.680,179.801,5.198,148.958
C01388=1107.641,-68.644,-48.668,179.801,5.192,148.957
C01389=1107.647,-68.894,-48.657,179.800,5.188,148.956
C01390=1107.652,-69.142,-48.646,179.800,5.183,148.955
C01391=1107.658,-69.393,-48.634,179.800,5.177,148.953
C01392=1107.662,-69.643,-48.623,179.801,5.172,148.952
C01393=1107.667,-69.892,-48.612,179.800,5.167,148.951
C01394=1107.673,-70.141,-48.600,179.800,5.162,148.950
C01395=1107.678,-70.391,-48.589,179.800,5.157,148.949
C01396=1107.683,-70.641,-48.577,179.801,5.152,148.948
C01397=1107.689,-70.891,-48.567,179.801,5.147,148.947
C01398=1107.693,-71.140,-48.556,179.800,5.142,148.946
C01399=1107.699,-71.390,-48.544,179.800,5.137,148.945
C01400=1107.703,-71.640,-48.533,179.801,5.132,148.943
C01401=1107.710,-71.890,-48.522,179.801,5.127,148.942
C01402=1107.713,-72.104,-48.512,179.800,5.122,148.941
C01403=1107.718,-72.318,-48.503,179.801,5.118,148.940
C01404=1107.723,-72.533,-48.493,179.801,5.113,148.939
C01405=1107.727,-72.748,-48.483,179.801,5.109,148.938
C01406=1107.732,-72.962,-48.473,179.801,5.104,148.937
C01407=1107.736,-73.177,-48.464,179.801,5.100,148.936
C01408=1107.741,-73.392,-48.455,179.801,5.096,148.935
C01409=1107.745,-73.606,-48.445,179.801,5.091,148.934
C01410=1107.750,-73.855,-48.434,179.801,5.086,148.933
C01411=1107.755,-74.105,-48.422,179.801,5.081,148.932
C01412=1107.761,-74.356,-48.411,179.801,5.076,148.931
C01413=1107.766,-74.604,-48.400,179.801,5.071,148.930
C01414=1107.771,-74.854,-48.389,179.801,5.066,148.929
C01415=1107.777,-75.105,-48.378,179.802,5.061,148.927
C01416=1107.782,-75.354,-48.367,179.801,5.055,148.926
C01417=1107.787,-75.604,-48.356,179.801,5.050,148.925
C01418=1107.792,-75.853,-48.345,179.801,5.044,148.924
C01419=1107.798,-76.103,-48.334,179.802,5.039,148.923
C01420=1107.803,-76.353,-48.323,179.802,5.034,148.922
C01421=1107.808,-76.602,-48.312,179.802,5.029,148.920
C01422=1107.814,-76.852,-48.301,179.802,5.024,148.919
C01423=1107.818,-77.102,-48.290,179.802,5.019,148.918
C01424=1107.824,-77.351,-48.279,179.802,5.014,148.917
C01425=1107.829,-77.601,-48.268,179.803,5.008,148.916
C01426=1107.834,-77.851,-48.256,179.803,5.003,148.915
C01427=1107.840,-78.101,-48.246,179.803,4.999,148.913
C01428=1107.844,-78.350,-48.235,179.804,4.994,148.912
C01429=1107.850,-78.600,-48.225,179.804,4.989,148.911
C01430=1107.855,-78.849,-48.213,179.804,4.984,148.910
C01431=1107.860,-79.100,-48.202,179.804,4.978,148.909
C01432=1107.866,-79.349,-48.191,179.804,4.973,148.908
C01433=1107.871,-79.599,-48.181,179.805,4.968,148.906
C01434=1107.876,-79.848,-48.170,179.805,4.963,148.905
C01435=1107.881,-80.098,-48.159,179.805,4.958,148.904
C01436=1107.887,-80.348,-48.148,179.805,4.952,148.903
C01437=1107.892,-80.598,-48.137,179.806,4.947,148.901
C01438=1107.897,-80.847,-48.126,179.806,4.942,148.900
C01439=1107.902,-81.097,-48.116,179.806,4.937,148.899
C01440=1107.907,-81.347,-48.105,179.806,4.932,148.898
C01441=1107.913,-81.596,-48.094,179.806,4.927,148.897
C01442=1107.918,-81.846,-48.083,179.806,4.921,148.896
C01443=1107.923,-82.095,-48.073,179.807,4.916,148.894
C01444=1107.929,-82.346,-48.061,179.807,4.912,148.893
C01445=1107.934,-82.595,-48.051,179.808,4.906,148.892
C01446=1107.939,-82.845,-48.040,179.808,4.901,148.891
C01447=1107.944,-83.095,-48.029,179.808,4.896,148.889
C01448=1107.949,-83.344,-48.018,179.808,4.891,148.888
C01449=1107.954,-83.594,-48.008,179.809,4.886,148.887
C01450=1107.960,-83.844,-47.998,179.809,4.881,148.886
C01451=1107.964,-84.094,-47.986,179.809,4.876,148.885
C01452=1107.970,-84.343,-47.976,179.809,4.870,148.883
C01453=1107.975,-84.593,-47.966,179.810,4.866,148.882
C01454=1107.980,-84.842,-47.955,179.810,4.861,148.881
C01455=1107.985,-85.093,-47.944,179.811,4.855,148.880
C01456=1107.992,-85.342,-47.933,179.811,4.850,148.879
C01457=1107.996,-85.592,-47.922,179.811,4.845,148.877
C01458=1108.001,-85.807,-47.914,179.811,4.841,148.876
C01459=1108.006,-86.021,-47.904,179.812,4.837,148.875
C01460=1108.010,-86.236,-47.895,179.812,4.832,148.874
C01461=1108.015,-86.451,-47.886,179.812,4.828,148.873
C01462=1108.019,-86.665,-47.877,179.813,4.824,148.872
C01463=1108.024,-86.880,-47.868,179.813,4.820,148.871
C01464=1108.027,-87.095,-47.859,179.813,4.815,148.870
C01465=1108.033,-87.309,-47.850,179.814,4.811,148.869
C01466=1108.038,-87.559,-47.839,179.814,4.806,148.868
C01467=1108.043,-87.808,-47.828,179.814,4.800,148.867
C01468=1108.049,-88.058,-47.818,179.815,4.796,148.866
C01469=1108.054,-88.308,-47.807,179.815,4.791,148.864
C01470=1108.059,-88.558,-47.797,179.816,4.785,148.863
C01471=1108.063,-88.807,-47.786,179.816,4.780,148.862
C01472=1108.069,-89.057,-47.776,179.817,4.776,148.861
C01473=1108.074,-89.307,-47.766,179.817,4.771,148.859
C01474=1108.079,-89.556,-47.755,179.817,4.766,148.858
C01475=1108.085,-89.806,-47.745,179.817,4.761,148.857
C01476=1108.090,-90.056,-47.735,179.818,4.756,148.856
C01477=1108.095,-90.305,-47.724,179.818,4.751,148.855
C01478=1108.100,-90.555,-47.713,179.818,4.746,148.853
C01479=1108.106,-90.805,-47.703,179.820,4.741,148.852
C01480=1108.111,-91.055,-47.692,179.820,4.736,148.851
C01481=1108.116,-91.305,-47.682,179.820,4.731,148.850
C01482=1108.122,-91.554,-47.672,179.820,4.726,148.848
C01483=1108.127,-91.805,-47.661,179.821,4.721,148.847
C01484=1108.133,-92.054,-47.651,179.821,4.716,148.846
C01485=1108.136,-92.303,-47.641,179.821,4.711,148.845
C01486=1108.142,-92.553,-47.630,179.822,4.707,148.844
C01487=1108.148,-92.802,-47.620,179.822,4.702,148.842
C01488=1108.153,-93.053,-47.610,179.823,4.697,148.841
C01489=1108.158,-93.302,-47.599,179.823,4.692,148.840
C01490=1108.163,-93.552,-47.589,179.824,4.687,148.839
C01491=1108.169,-93.802,-47.579,179.824,4.683,148.838
C01492=1108.174,-94.052,-47.568,179.825,4.677,148.836
C01493=1108.179,-94.302,-47.558,179.825,4.672,148.835
C01494=1108.184,-94.551,-47.548,179.826,4.668,148.834
C01495=1108.190,-94.801,-47.538,179.826,4.662,148.833
C01496=1108.195,-95.051,-47.527,179.826,4.657,148.832
C01497=1108.201,-95.300,-47.517,179.827,4.653,148.830
C01498=1108.206,-95.550,-47.507,179.827,4.648,148.829
C01499=1108.211,-95.800,-47.496,179.827,4.643,148.828
C01500=1108.216,-96.049,-47.487,179.827,4.638,148.827
C01501=1108.221,-96.300,-47.476,179.828,4.634,148.826
C01502=1108.227,-96.549,-47.466,179.828,4.628,148.825
C01503=1108.232,-96.799,-47.456,179.829,4.623,148.823
C01504=1108.237,-97.049,-47.445,179.829,4.619,148.822
C01505=1108.242,-97.298,-47.436,179.830,4.614,148.821
C01506=1108.248,-97.548,-47.425,179.830,4.609,148.820
C01507=1108.253,-97.797,-47.415,179.831,4.604,148.819
C01508=1108.258,-98.048,-47.405,179.831,4.599,148.817
C01509=1108.264,-98.297,-47.394,179.831,4.594,148.816
C01510=1108.269,-98.546,-47.385,179.831,4.589,148.815
C01511=1108.274,-98.797,-47.374,179.832,4.585,148.814
C01512=1108.280,-99.047,-47.365,179.832,4.579,148.813
C01513=1108.285,-99.296,-47.354,179.832,4.574,148.811
C01514=1108.289,-99.511,-47.346,179.833,4.570,148.810
C01515=1108.293,-99.725,-47.337,179.834,4.566,148.809
C01516=1108.299,-99.940,-47.328,179.834,4.562,148.808
C01517=1108.303,-100.155,-47.319,179.834,4.557,148.807
C01518=1108.307,-100.370,-47.311,179.834,4.553,148.806
C01519=1108.311,-100.584,-47.302,179.835,4.549,148.805
C01520=1108.317,-100.799,-47.294,179.835,4.545,148.804
C01521=1108.321,-101.013,-47.285,179.836,4.541,148.803
C01522=1108.326,-101.264,-47.275,179.836,4.535,148.802
C01523=1108.331,-101.513,-47.265,179.836,4.530,148.801
C01524=1108.337,-101.763,-47.256,179.836,4.525,148.800
C01525=1108.342,-102.013,-47.245,179.837,4.521,148.798
C01526=1108.347,-102.263,-47.235,179.837,4.516,148.797
C01527=1108.352,-102.512,-47.225,179.838,4.510,148.796
C01528=1108.358,-102.762,-47.215,179.838,4.505,148.795
C01529=1108.363,-103.012,-47.206,179.839,4.501,148.794
C01530=1108.368,-103.262,-47.195,179.839,4.496,148.792
C01531=1108.374,-103.511,-47.185,179.839,4.491,148.791
C01532=1108.379,-103.760,-47.176,179.839,4.486,148.790
C01533=1108.384,-104.011,-47.166,179.840,4.480,148.789
C01534=1108.390,-104.261,-47.156,179.840,4.476,148.788
C01535=1108.394,-104.510,-47.146,179.841,4.471,148.786
C01536=1108.400,-104.760,-47.136,179.841,4.466,148.785
C01537=1108.406,-105.010,-47.126,179.841,4.461,148.784
C01538=1108.410,-105.260,-47.116,179.842,4.456,148.783
C01539=1108.416,-105.509,-47.106,179.842,4.451,148.782
C01540=1108.421,-105.759,-47.096,179.843,4.446,148.780
C01541=1108.427,-106.009,-47.087,179.843,4.440,148.779
C01542=1108.432,-106.258,-47.077,179.843,4.435,148.778
C01543=1108.436,-106.508,-47.067,179.844,4.431,148.776
C01544=1108.442,-106.758,-47.057,179.844,4.426,148.775
C01545=1108.447,-107.008,-47.048,179.845,4.421,148.774
C01546=1108.453,-107.257,-47.037,179.845,4.415,148.773
C01547=1108.458,-107.507,-47.029,179.846,4.411,148.772
C01548=1108.463,-107.757,-47.018,179.846,4.406,148.770
C01549=1108.469,-108.007,-47.008,179.846,4.401,148.769
C01550=1108.474,-108.257,-46.999,179.847,4.396,148.768
C01551=1108.479,-108.506,-46.989,179.847,4.390,148.767
C01552=1108.484,-108.756,-46.980,179.847,4.385,148.766
C01553=1108.490,-109.006,-46.970,179.848,4.381,148.764
C01554=1108.494,-109.255,-46.960,179.849,4.375,148.763
C01555=1108.500,-109.506,-46.950,179.849,4.370,148.762
C01556=1108.505,-109.755,-46.940,179.849,4.365,148.761
C01557=1108.511,-110.005,-46.931,179.849,4.360,148.759
C01558=1108.516,-110.254,-46.921,179.850,4.356,148.758
C01559=1108.522,-110.504,-46.912,179.850,4.350,148.757
C01560=1108.527,-110.754,-46.902,179.851,4.345,148.756
C01561=1108.532,-111.004,-46.892,179.851,4.340,148.755
C01562=1108.537,-111.254,-46.883,179.852,4.335,148.753
C01563=1108.542,-111.503,-46.873,179.852,4.329,148.752
C01564=1108.548,-111.753,-46.864,179.852,4.324,148.751
C01565=1108.553,-112.003,-46.853,179.853,4.320,148.749
C01566=1108.558,-112.253,-46.845,179.853,4.315,148.748
C01567=1108.564,-112.502,-46.834,179.854,4.310,148.747
C01568=1108.569,-112.752,-46.825,179.854,4.304,148.746
C01569=1108.575,-113.001,-46.815,179.854,4.299,148.745
C01570=1108.579,-113.217,-46.807,179.855,4.295,148.743
C01571=1108.583,-113.432,-46.799,179.855,4.291,148.742
C01572=1108.588,-113.646,-46.791,179.856,4.286,148.741
C01573=1108.593,-113.861,-46.783,179.856,4.282,148.740
C01574=1108.597,-114.076,-46.775,179.857,4.278,148.739
C01575=1108.602,-114.290,-46.766,179.856,4.273,148.738
C01576=1108.607,-114.505,-46.759,179.857,4.268,148.737
C01577=1108.610,-114.721,-46.750,179.858,4.264,148.736
C01578=1108.616,-114.971,-46.741,179.858,4.259,148.735
C01579=1108.621,-115.220,-46.731,179.858,4.254,148.734
C01580=1108.626,-115.470,-46.722,179.859,4.249,148.732
C01581=1108.632,-115.719,-46.712,179.859,4.243,148.731
C01582=1108.637,-115.969,-46.703,179.859,4.238,148.730
C01583=1108.643,-116.219,-46.693,179.860,4.233,148.728
C01584=1108.648,-116.469,-46.684,179.860,4.228,148.727
C01585=1108.653,-116.718,-46.675,179.861,4.222,148.726
C01586=1108.659,-116.968,-46.665,179.861,4.217,148.725
C01587=1108.664,-117.218,-46.656,179.861,4.212,148.723
C01588=1108.670,-117.468,-46.646,179.862,4.208,148.722
C01589=1108.675,-117.717,-46.637,179.863,4.202,148.721
C01590=1108.680,-117.967,-46.628,179.863,4.197,148.719
C01591=1108.686,-118.217,-46.618,179.864,4.192,148.718
C01592=1108.691,-118.466,-46.609,179.864,4.187,148.717
C01593=1108.696,-118.716,-46.600,179.865,4.181,148.716
C01594=1108.702,-118.966,-46.590,179.865,4.176,148.714
C01595=1108.707,-119.216,-46.581,179.865,4.171,148.713
C01596=1108.712,-119.466,-46.572,179.865,4.166,148.712
C01597=1108.717,-119.715,-46.563,179.866,4.160,148.710
C01598=1108.723,-119.966,-46.553,179.867,4.155,148.709
C01599=1108.728,-120.215,-46.544,179.867,4.150,148.708
C01600=1108.733,-120.465,-46.535,179.868,4.144,148.707
C01601=1108.739,-120.715,-46.525,179.868,4.139,148.705
C01602=1108.744,-120.965,-46.517,179.868,4.134,148.704
C01603=1108.749,-121.214,-46.508,179.869,4.128,148.703
C01604=1108.754,-121.464,-46.498,179.869,4.123,148.701
C01605=1108.760,-121.714,-46.489,179.870,4.118,148.700
C01606=1108.765,-121.964,-46.480,179.870,4.113,148.699
C01607=1108.770,-122.214,-46.471,179.871,4.107,148.698
C01608=1108.775,-122.463,-46.461,179.871,4.102,148.696
C01609=1108.781,-122.713,-46.452,179.872,4.097,148.695
C01610=1108.786,-122.963,-46.443,179.872,4.092,148.694
C01611=1108.791,-123.213,-46.434,179.872,4.086,148.692
C01612=1108.796,-123.463,-46.425,179.873,4.081,148.691
C01613=1108.802,-123.713,-46.415,179.873,4.076,148.690
C01614=1108.807,-123.962,-46.406,179.874,4.071,148.689
C01615=1108.813,-124.211,-46.397,179.875,4.065,148.687
C01616=1108.818,-124.461,-46.388,179.875,4.060,148.686
C01617=1108.823,-124.711,-46.379,179.876,4.054,148.684
C01618=1108.829,-124.961,-46.370,179.876,4.049,148.683
C01619=1108.834,-125.211,-46.361,179.876,4.044,148.682
C01620=1108.839,-125.461,-46.352,179.877,4.038,148.680
C01621=1108.845,-125.711,-46.343,179.877,4.033,148.679
C01622=1108.850,-125.960,-46.334,179.878,4.028,148.678
C01623=1108.855,-126.210,-46.325,179.878,4.023,148.677
C01624=1108.861,-126.460,-46.315,179.879,4.017,148.675
C01625=1108.866,-126.710,-46.306,179.880,4.012,148.674
C01626=1108.871,-126.925,-46.299,179.880,4.007,148.673
C01627=1108.875,-127.139,-46.292,179.881,4.002,148.671
C01628=1108.879,-127.355,-46.284,179.881,3.998,148.670
C01629=1108.884,-127.569,-46.276,179.881,3.993,148.669
C01630=1108.889,-127.784,-46.268,179.882,3.988,148.668
C01631=1108.894,-127.999,-46.261,179.882,3.984,148.667
C01632=1108.898,-128.214,-46.254,179.882,3.979,148.666
C01633=1108.902,-128.428,-46.245,179.883,3.975,148.665
C01634=1108.479,-128.419,-46.272,179.890,3.978,148.663
C01635=1108.475,-128.204,-46.279,179.890,3.983,148.664
C01636=1108.471,-127.989,-46.286,179.889,3.988,148.666
C01637=1108.466,-127.775,-46.295,179.889,3.993,148.667
C01638=1108.461,-127.560,-46.302,179.888,3.997,148.668
C01639=1108.456,-127.345,-46.310,179.888,4.002,148.669
C01640=1108.452,-127.130,-46.317,179.887,4.006,148.670
C01641=1108.447,-126.915,-46.326,179.887,4.011,148.671
C01642=1108.443,-126.700,-46.333,179.887,4.015,148.672
C01643=1108.437,-126.450,-46.342,179.886,4.021,148.674
C01644=1108.432,-126.200,-46.351,179.886,4.026,148.675
C01645=1108.427,-125.950,-46.360,179.885,4.032,148.677
C01646=1108.422,-125.701,-46.369,179.885,4.038,148.678
C01647=1108.417,-125.451,-46.378,179.884,4.043,148.679
C01648=1108.411,-125.201,-46.388,179.884,4.048,148.680
C01649=1108.406,-124.951,-46.397,179.883,4.054,148.682
C01650=1108.401,-124.702,-46.406,179.883,4.059,148.683
C01651=1108.395,-124.452,-46.415,179.883,4.064,148.684
C01652=1108.390,-124.203,-46.423,179.882,4.070,148.686
C01653=1108.384,-123.952,-46.433,179.881,4.075,148.687
C01654=1108.379,-123.703,-46.442,179.881,4.080,148.689
C01655=1108.374,-123.453,-46.451,179.880,4.086,148.690
C01656=1108.369,-123.203,-46.460,179.880,4.091,148.691
C01657=1108.363,-122.953,-46.470,179.879,4.096,148.692
C01658=1108.357,-122.703,-46.479,179.879,4.101,148.694
C01659=1108.353,-122.454,-46.488,179.879,4.107,148.695
C01660=1108.347,-122.204,-46.497,179.878,4.112,148.696
C01661=1108.341,-121.954,-46.507,179.878,4.117,148.698
C01662=1108.336,-121.704,-46.515,179.877,4.122,148.699
C01663=1108.331,-121.455,-46.525,179.876,4.128,148.700
C01664=1108.326,-121.205,-46.534,179.876,4.133,148.701
C01665=1108.320,-120.955,-46.543,179.876,4.138,148.703
C01666=1108.315,-120.705,-46.552,179.875,4.144,148.704
C01667=1108.310,-120.456,-46.562,179.875,4.149,148.705
C01668=1108.304,-120.206,-46.571,179.875,4.154,148.707
C01669=1108.299,-119.956,-46.580,179.874,4.160,148.708
C01670=1108.294,-119.706,-46.589,179.873,4.164,148.709
C01671=1108.289,-119.457,-46.599,179.873,4.169,148.710
C01672=1108.283,-119.207,-46.608,179.872,4.175,148.712
C01673=1108.278,-118.957,-46.617,179.871,4.180,148.713
C01674=1108.273,-118.707,-46.627,179.871,4.185,148.714
C01675=1108.267,-118.458,-46.636,179.871,4.190,148.716
C01676=1108.262,-118.208,-46.645,179.870,4.196,148.717
C01677=1108.257,-117.958,-46.655,179.870,4.201,148.718
C01678=1108.252,-117.708,-46.664,179.870,4.206,148.719
C01679=1108.246,-117.458,-46.673,179.869,4.211,148.721
C01680=1108.241,-117.209,-46.683,179.869,4.217,148.722
C01681=1108.236,-116.959,-46.692,179.868,4.222,148.723
C01682=1108.230,-116.709,-46.703,179.868,4.227,148.725
C01683=1108.225,-116.460,-46.711,179.868,4.232,148.726
C01684=1108.220,-116.210,-46.720,179.866,4.237,148.727
C01685=1108.215,-115.960,-46.731,179.866,4.242,148.728
C01686=1108.209,-115.710,-46.740,179.866,4.247,148.730
C01687=1108.204,-115.460,-46.750,179.866,4.252,148.731
C01688=1108.199,-115.210,-46.759,179.865,4.258,148.732
C01689=1108.194,-114.961,-46.769,179.864,4.263,148.733
C01690=1108.188,-114.711,-46.778,179.864,4.268,148.735
C01691=1108.183,-114.496,-46.786,179.864,4.272,148.736
C01692=1108.179,-114.281,-46.794,179.863,4.277,148.737
C01693=1108.174,-114.067,-46.802,179.863,4.281,148.738
C01694=1108.170,-113.852,-46.811,179.862,4.286,148.739
C01695=1108.166,-113.637,-46.819,179.862,4.290,148.740
C01696=1108.161,-113.422,-46.827,179.862,4.295,148.741
C01697=1108.156,-113.208,-46.835,179.862,4.299,148.742
C01698=1108.152,-112.993,-46.844,179.861,4.303,148.743
C01699=1108.146,-112.743,-46.853,179.860,4.308,148.745
C01700=1108.141,-112.494,-46.863,179.860,4.313,148.746
C01701=1108.135,-112.244,-46.872,179.860,4.319,148.747
C01702=1108.130,-111.994,-46.882,179.860,4.324,148.748
C01703=1108.125,-111.744,-46.892,179.859,4.329,148.749
C01704=1108.120,-111.494,-46.901,179.859,4.334,148.751
C01705=1108.114,-111.244,-46.911,179.858,4.338,148.752
C01706=1108.109,-110.995,-46.920,179.858,4.344,148.753
C01707=1108.104,-110.745,-46.931,179.857,4.349,148.755
C01708=1108.099,-110.496,-46.939,179.857,4.354,148.756
C01709=1108.093,-110.246,-46.950,179.857,4.359,148.757
C01710=1108.089,-109.995,-46.959,179.857,4.365,148.758
C01711=1108.083,-109.746,-46.969,179.856,4.369,148.759
C01712=1108.078,-109.496,-46.978,179.855,4.374,148.761
C01713=1108.072,-109.246,-46.988,179.855,4.379,148.762
C01714=1108.067,-108.997,-46.998,179.854,4.385,148.763
C01715=1108.061,-108.747,-47.007,179.854,4.390,148.764
C01716=1108.056,-108.497,-47.018,179.853,4.394,148.766
C01717=1108.052,-108.248,-47.028,179.853,4.399,148.767
C01718=1108.046,-107.997,-47.037,179.853,4.405,148.768
C01719=1108.041,-107.748,-47.047,179.853,4.410,148.769
C01720=1108.035,-107.499,-47.057,179.852,4.415,148.770
C01721=1108.029,-107.249,-47.066,179.852,4.419,148.772
C01722=1108.025,-106.999,-47.076,179.851,4.424,148.773
C01723=1108.019,-106.749,-47.087,179.851,4.430,148.774
C01724=1108.014,-106.499,-47.095,179.851,4.435,148.775
C01725=1108.009,-106.250,-47.106,179.851,4.440,148.776
C01726=1108.004,-105.999,-47.116,179.850,4.444,148.778
C01727=1107.999,-105.750,-47.126,179.849,4.450,148.779
C01728=1107.993,-105.500,-47.135,179.849,4.455,148.780
C01729=1107.987,-105.250,-47.146,179.849,4.460,148.781
C01730=1107.982,-105.001,-47.155,179.848,4.464,148.783
C01731=1107.977,-104.751,-47.166,179.848,4.470,148.784
C01732=1107.972,-104.501,-47.175,179.847,4.475,148.785
C01733=1107.967,-104.252,-47.185,179.847,4.480,148.786
C01734=1107.961,-104.002,-47.195,179.847,4.485,148.787
C01735=1107.957,-103.752,-47.205,179.846,4.489,148.789
C01736=1107.951,-103.502,-47.215,179.846,4.494,148.790
C01737=1107.945,-103.252,-47.225,179.846,4.500,148.791
C01738=1107.940,-103.003,-47.234,179.845,4.505,148.792
C01739=1107.935,-102.753,-47.245,179.845,4.509,148.793
C01740=1107.930,-102.503,-47.255,179.844,4.514,148.795
C01741=1107.925,-102.254,-47.264,179.844,4.519,148.796
C01742=1107.919,-102.004,-47.274,179.844,4.525,148.797
C01743=1107.914,-101.754,-47.285,179.843,4.529,148.798
C01744=1107.908,-101.504,-47.295,179.843,4.534,148.799
C01745=1107.904,-101.255,-47.305,179.843,4.539,148.801
C01746=1107.899,-101.005,-47.315,179.842,4.544,148.802
C01747=1107.894,-100.790,-47.324,179.842,4.549,148.803
C01748=1107.889,-100.575,-47.332,179.841,4.553,148.804
C01749=1107.884,-100.361,-47.341,179.841,4.557,148.805
C01750=1107.880,-100.146,-47.350,179.841,4.561,148.806
C01751=1107.876,-99.931,-47.358,179.840,4.566,148.807
C01752=1107.871,-99.717,-47.367,179.840,4.570,148.808
C01753=1107.866,-99.502,-47.375,179.840,4.574,148.809
C01754=1107.862,-99.287,-47.384,179.839,4.578,148.810
C01755=1107.857,-99.037,-47.394,179.839,4.583,148.811
C01756=1107.851,-98.788,-47.404,179.839,4.588,148.813
C01757=1107.846,-98.538,-47.415,179.838,4.593,148.814
C01758=1107.840,-98.288,-47.425,179.838,4.598,148.815
C01759=1107.836,-98.039,-47.435,179.837,4.603,148.816
C01760=1107.831,-97.789,-47.445,179.837,4.607,148.817
C01761=1107.825,-97.539,-47.455,179.836,4.612,148.819
C01762=1107.819,-97.290,-47.466,179.836,4.618,148.820
C01763=1107.814,-97.039,-47.476,179.836,4.623,148.821
C01764=1107.810,-96.790,-47.486,179.835,4.627,148.822
C01765=1107.804,-96.540,-47.496,179.835,4.632,148.823
C01766=1107.799,-96.290,-47.507,179.835,4.637,148.825
C01767=1107.793,-96.041,-47.517,179.834,4.642,148.826
C01768=1107.788,-95.791,-47.527,179.834,4.647,148.827
C01769=1107.783,-95.541,-47.538,179.834,4.652,148.828
C01770=1107.778,-95.292,-47.547,179.833,4.657,148.829
C01771=1107.772,-95.042,-47.557,179.833,4.661,148.831
C01772=1107.767,-94.792,-47.568,179.832,4.667,148.832
C01773=1107.762,-94.542,-47.578,179.832,4.672,148.833
C01774=1107.757,-94.292,-47.589,179.831,4.676,148.834
C01775=1107.751,-94.043,-47.599,179.831,4.681,148.835
C01776=1107.746,-93.793,-47.609,179.831,4.686,148.836
C01777=1107.741,-93.543,-47.620,179.830,4.691,148.838
C01778=1107.736,-93.294,-47.630,179.830,4.696,148.839
C01779=1107.731,-93.044,-47.641,179.829,4.700,148.840
C01780=1107.725,-92.794,-47.651,179.829,4.705,148.841
C01781=1107.720,-92.545,-47.661,179.829,4.711,148.842
C01782=1107.715,-92.295,-47.672,179.828,4.715,148.844
C01783=1107.709,-92.045,-47.682,179.828,4.720,148.845
C01784=1107.704,-91.795,-47.692,179.828,4.725,148.846
C01785=1107.699,-91.545,-47.703,179.827,4.730,148.847
C01786=1107.693,-91.296,-47.714,179.827,4.735,148.848
C01787=1107.688,-91.046,-47.724,179.826,4.740,148.850
C01788=1107.683,-90.797,-47.734,179.826,4.745,148.851
C01789=1107.678,-90.546,-47.745,179.825,4.750,148.852
C01790=1107.673,-90.297,-47.755,179.825,4.755,148.853
C01791=1107.668,-90.047,-47.765,179.825,4.760,148.855
C01792=1107.663,-89.798,-47.776,179.824,4.764,148.856
C01793=1107.658,-89.548,-47.787,179.824,4.769,148.857
C01794=1107.652,-89.298,-47.797,179.823,4.775,148.858
C01795=1107.646,-89.049,-47.807,179.823,4.780,148.859
C01796=1107.641,-88.798,-47.818,179.822,4.784,148.861
C01797=1107.636,-88.549,-47.828,179.822,4.789,148.862
C01798=1107.631,-88.299,-47.839,179.822,4.795,148.863
C01799=1107.625,-88.050,-47.849,179.821,4.800,148.864
C01800=1107.620,-87.799,-47.860,179.821,4.805,148.865
C01801=1107.615,-87.550,-47.871,179.820,4.809,148.867
C01802=1107.610,-87.300,-47.881,179.820,4.815,148.868
C01803=1107.605,-87.085,-47.890,179.820,4.818,148.869
C01804=1107.601,-86.871,-47.900,179.820,4.824,148.870
C01805=1107.596,-86.656,-47.909,179.819,4.828,148.871
C01806=1107.592,-86.442,-47.918,179.819,4.832,148.872
C01807=1107.587,-86.227,-47.927,179.818,4.836,148.873
C01808=1107.583,-86.013,-47.936,179.819,4.841,148.874
C01809=1107.578,-85.797,-47.945,179.818,4.845,148.875
C01810=1107.574,-85.584,-47.954,179.818,4.849,148.876
C01811=1107.569,-85.334,-47.965,179.818,4.854,148.877
C01812=1107.564,-85.084,-47.975,179.817,4.859,148.878
C01813=1107.558,-84.834,-47.987,179.817,4.865,148.880
C01814=1107.553,-84.584,-47.997,179.817,4.870,148.881
C01815=1107.548,-84.334,-48.008,179.816,4.875,148.882
C01816=1107.542,-84.085,-48.019,179.816,4.879,148.883
C01817=1107.537,-83.835,-48.029,179.815,4.885,148.885
C01818=1107.532,-83.586,-48.040,179.815,4.890,148.886
C01819=1107.527,-83.336,-48.051,179.815,4.895,148.887
C01820=1107.521,-83.086,-48.061,179.815,4.900,148.888
C01821=1107.517,-82.837,-48.072,179.815,4.905,148.889
C01822=1107.511,-82.587,-48.082,179.814,4.911,148.891
C01823=1107.506,-82.337,-48.094,179.814,4.916,148.892
C01824=1107.500,-82.088,-48.105,179.814,4.921,148.893
C01825=1107.495,-81.837,-48.115,179.813,4.925,148.894
C01826=1107.490,-81.588,-48.126,179.813,4.930,148.895
C01827=1107.485,-81.338,-48.137,179.813,4.936,148.897
C01828=1107.480,-81.088,-48.148,179.812,4.941,148.898
C01829=1107.475,-80.839,-48.158,179.812,4.946,148.899
C01830=1107.469,-80.589,-48.170,179.812,4.951,148.900
C01831=1107.463,-80.339,-48.180,179.812,4.956,148.901
C01832=1107.459,-80.090,-48.192,179.812,4.961,148.903
C01833=1107.454,-79.840,-48.202,179.812,4.966,148.904
C01834=1107.449,-79.591,-48.213,179.811,4.972,148.905
C01835=1107.443,-79.340,-48.224,179.811,4.977,148.906
C01836=1107.437,-79.091,-48.235,179.811,4.982,148.908
C01837=1107.432,-78.841,-48.246,179.811,4.987,148.909
C01838=1107.428,-78.591,-48.257,179.810,4.992,148.910
C01839=1107.422,-78.342,-48.267,179.810,4.998,148.911
C01840=1107.417,-78.092,-48.279,179.810,5.003,148.912
C01841=1107.411,-77.842,-48.289,179.810,5.008,148.913
C01842=1107.406,-77.593,-48.301,179.810,5.013,148.915
C01843=1107.402,-77.343,-48.312,179.810,5.018,148.916
C01844=1107.395,-77.093,-48.323,179.809,5.023,148.917
